KUKA KRL program: f1_Kuka_APT213T02S13.SRC

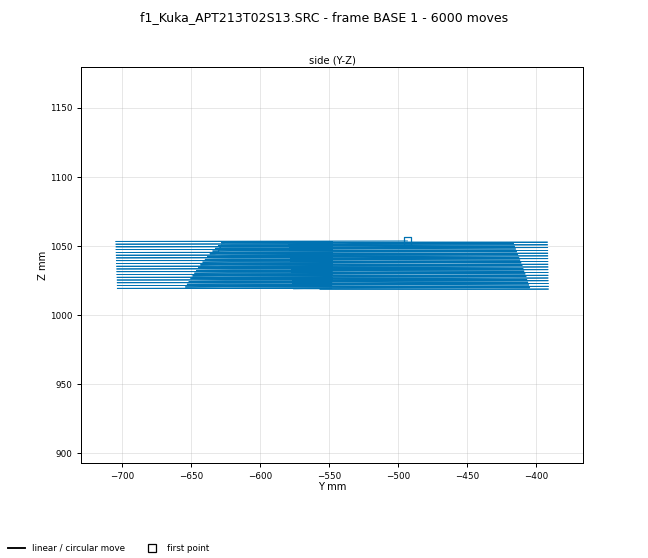
[picture p0: tool path of f1_Kuka_APT213T02S13.SRC in frame BASE 1, 6000 of 6001 moves have a stored position in this frame; points joined in program order, loops and branches not executed]
&ACCESS RVP
&REL 2
&PARAM TEMPLATE = C:\KRC\Roboter\Template\vorgabe
&PARAM EDITMASK = *
DEF f1_Kuka_APT213T02S13()


;FOLD INI;%{PE}%V3.2.0,%MKUKATPBASIS,%CINIT,%VCOMMON,%P
  ;FOLD BAS INI;%{E}%V3.2.0,%MKUKATPBASIS,%CINIT,%VINIT,%P
    GLOBAL INTERRUPT DECL 3 WHEN $STOPMESS==TRUE DO IR_STOPM ( )
    INTERRUPT ON 3
    BAS (#INITMOV,0 )
  ;ENDFOLD (BAS INI)
  ;FOLD USER INI;%{E}%V3.2.0,%MKUKATPUSER,%CINIT,%VINIT,%P
    ;Make your modifications here
  ;ENDFOLD (USER INI)
;ENDFOLD (INI)


;*** Make Null PTP Move
  PTP $pos_act

;*** Auto Load The Correct TOOL Data
  $tool=tool_data[2]

;*** Auto Load The Correct BASE Data
  $base=base_data[1]

  $ADVANCE = 5

;*** Restate Last Velocity
MMPM(30000.0)
SetRPM(8000)
LIN {X 0.196,Y -493.060,Z 1053.803,A 0.000,B 0.000,C 90.000,E1 180.573} C_DIS
LIN {X -0.057,Y -499.392,Z 1053.797,A 0.000,B 0.000,C 90.000,E1 179.542} C_DIS
LIN {X 0.076,Y -508.774,Z 1053.788,A 0.000,B 0.000,C 90.000,E1 177.879} C_DIS
LIN {X 0.040,Y -514.640,Z 1053.783,A 0.000,B 0.000,C 90.000,E1 176.846} C_DIS
LIN {X 0.239,Y -524.434,Z 1053.773,A 0.000,B 0.000,C 90.000,E1 175.065} C_DIS
LIN {X -0.105,Y -531.617,Z 1053.766,A 0.000,B 0.000,C 90.000,E1 173.799} C_DIS
LIN {X -0.076,Y -537.841,Z 1053.759,A 0.000,B 0.000,C 90.000,E1 172.648} C_DIS
LIN {X 0.196,Y -545.614,Z 1053.751,A 0.000,B 0.000,C 90.000,E1 171.197} C_DIS
LIN {X 0.075,Y -553.106,Z 1053.743,A 0.000,B 0.000,C 90.000,E1 169.803} C_DIS
LIN {X -0.212,Y -559.744,Z 1053.736,A 0.000,B 0.000,C 90.000,E1 168.578} C_DIS
LIN {X -0.238,Y -567.509,Z 1053.728,A 0.000,B 0.000,C 90.000,E1 167.061} C_DIS
LIN {X -0.052,Y -573.559,Z 1053.721,A 0.000,B 0.000,C 90.000,E1 165.811} C_DIS
LIN {X 0.098,Y -579.321,Z 1053.714,A 0.000,B 0.000,C 90.000,E1 164.574} C_DIS
LIN {X 0.012,Y -584.212,Z 1053.708,A 0.000,B 0.000,C 90.000,E1 163.504} C_DIS
LIN {X -0.002,Y -587.133,Z 1053.705,A 0.000,B 0.000,C 90.000,E1 162.834} C_DIS
LIN {X 0.006,Y -591.638,Z 1053.699,A 0.000,B 0.000,C 90.000,E1 161.764} C_DIS
LIN {X 0.001,Y -594.742,Z 1053.694,A 0.000,B 0.000,C 90.000,E1 160.967} C_DIS
LIN {X -0.165,Y -597.776,Z 1053.690,A 0.000,B 0.000,C 90.000,E1 160.188} C_DIS
LIN {X -0.189,Y -601.641,Z 1053.684,A 0.000,B 0.000,C 90.000,E1 159.135} C_DIS
LIN {X 0.188,Y -605.246,Z 1053.678,A 0.000,B 0.000,C 90.000,E1 158.050} C_DIS
LIN {X 0.000,Y -607.751,Z 1053.674,A 0.000,B 0.000,C 90.000,E1 157.283} C_DIS
LIN {X 0.082,Y -611.784,Z 1053.667,A 0.000,B 0.000,C 90.000,E1 155.973} C_DIS
LIN {X 0.223,Y -615.402,Z 1053.659,A 0.000,B 0.000,C 90.000,E1 154.665} C_DIS
LIN {X 0.159,Y -617.516,Z 1053.655,A 0.000,B 0.000,C 90.000,E1 153.896} C_DIS
LIN {X 0.107,Y -620.213,Z 1053.649,A 0.000,B 0.000,C 90.000,E1 152.871} C_DIS
LIN {X 0.086,Y -623.401,Z 1053.642,A 0.000,B 0.000,C 90.000,E1 151.591} C_DIS
LIN {X -0.142,Y -625.870,Z 1053.637,A 0.000,B 0.000,C 90.000,E1 150.589} C_DIS
LIN {X 0.226,Y -628.970,Z 1053.630,A 0.000,B 0.000,C 90.000,E1 149.282} C_DIS
LIN {X -0.091,Y -632.383,Z 1053.621,A 0.000,B 0.000,C 90.000,E1 147.788} C_DIS
LIN {X -0.338,Y -635.741,Z 1053.613,A 0.000,B 0.000,C 90.000,E1 146.294} C_DIS
LIN {X 0.223,Y -639.581,Z 1053.603,A 0.000,B 0.000,C 90.000,E1 144.482} C_DIS
LIN {X -0.163,Y -643.368,Z 1053.593,A 0.000,B 0.000,C 90.000,E1 142.763} C_DIS
LIN {X 0.016,Y -646.627,Z 1053.585,A 0.000,B 0.000,C 90.000,E1 141.251} C_DIS
LIN {X 0.163,Y -649.847,Z 1053.577,A 0.000,B 0.000,C 90.000,E1 139.747} C_DIS
LIN {X 0.329,Y -653.619,Z 1053.567,A 0.000,B 0.000,C 90.000,E1 138.000} C_DIS
LIN {X 0.123,Y -656.954,Z 1053.559,A 0.000,B 0.000,C 90.000,E1 136.539} C_DIS
LIN {X -0.151,Y -665.082,Z 1053.541,A 0.000,B 0.000,C 90.000,E1 133.380} C_DIS
LIN {X -0.134,Y -668.997,Z 1053.533,A 0.000,B 0.000,C 90.000,E1 131.919} C_DIS
LIN {X -0.029,Y -673.558,Z 1053.523,A 0.000,B 0.000,C 90.000,E1 130.216} C_DIS
LIN {X 0.230,Y -677.442,Z 1053.515,A 0.000,B 0.000,C 90.000,E1 128.749} C_DIS
LIN {X 0.011,Y -680.552,Z 1053.509,A 0.000,B 0.000,C 90.000,E1 127.569} C_DIS
LIN {X -0.011,Y -684.183,Z 1053.501,A 0.000,B 0.000,C 90.000,E1 126.137} C_DIS
LIN {X 0.008,Y -687.232,Z 1053.494,A 0.000,B 0.000,C 90.000,E1 124.945} C_DIS
LIN {X -0.079,Y -691.303,Z 1053.485,A 0.000,B 0.000,C 90.000,E1 123.293} C_DIS
LIN {X 0.024,Y -693.615,Z 1053.480,A 0.000,B 0.000,C 90.000,E1 122.339} C_DIS
LIN {X 0.155,Y -695.792,Z 1053.474,A 0.000,B 0.000,C 90.000,E1 121.386} C_DIS
LIN {X -0.048,Y -697.830,Z 1053.469,A 0.000,B 0.000,C 90.000,E1 120.463} C_DIS
LIN {X -0.222,Y -699.569,Z 1053.464,A 0.000,B 0.000,C 90.000,E1 119.539} C_DIS
LIN {X -0.034,Y -700.589,Z 1053.460,A 0.000,B 0.000,C 90.000,E1 118.821} C_DIS
LIN {X -0.015,Y -702.523,Z 1053.450,A 0.000,B 0.000,C 90.000,E1 116.950} C_DIS
LIN {X -0.150,Y -703.521,Z 1053.445,A 0.000,B 0.000,C 90.000,E1 116.027} C_DIS
LIN {X 0.042,Y -704.221,Z 1053.439,A 0.000,B 0.000,C 90.000,E1 115.079} C_DIS
LIN {X -0.324,Y -704.422,Z 1053.437,A 0.000,B 0.000,C 90.000,E1 114.643} C_DIS
LIN {X -0.045,Y -704.190,Z 1053.434,A 0.000,B 0.000,C 90.000,E1 114.155} C_DIS
LIN {X 0.240,Y -703.803,Z 1053.433,A 0.000,B 0.000,C 90.000,E1 113.898} C_DIS
LIN {X -0.123,Y -702.567,Z 1053.430,A 0.000,B 0.000,C 90.000,E1 113.462} C_DIS
LIN {X 0.017,Y -702.065,Z 1053.430,A 0.000,B 0.000,C 90.000,E1 113.334} C_DIS
LIN {X -0.357,Y -698.967,Z 1053.427,A 0.000,B 0.000,C 90.000,E1 112.898} C_DIS
LIN {X -0.223,Y -698.087,Z 1053.426,A 0.000,B 0.000,C 90.000,E1 112.770} C_DIS
LIN {X -0.093,Y -696.802,Z 1053.426,A 0.000,B 0.000,C 90.000,E1 112.642} C_DIS
LIN {X 0.037,Y -694.773,Z 1053.425,A 0.000,B 0.000,C 90.000,E1 112.514} C_DIS
LIN {X -0.179,Y -687.842,Z 1053.423,A 0.000,B 0.000,C 90.000,E1 112.206} C_DIS
LIN {X 0.203,Y -685.670,Z 1053.423,A 0.000,B 0.000,C 90.000,E1 112.099} C_DIS
LIN {X 0.017,Y -684.206,Z 1053.423,A 0.000,B 0.000,C 90.000,E1 112.078} C_DIS
LIN {X 0.020,Y -675.787,Z 1053.422,A 0.000,B 0.000,C 90.000,E1 111.972} C_DIS
LIN {X -0.030,Y -609.618,Z 1053.422,A 0.000,B 0.000,C 90.000,E1 111.972} C_DIS
LIN {X -0.052,Y -604.028,Z 1053.421,A 0.000,B 0.000,C 90.000,E1 111.770} C_DIS
LIN {X -0.108,Y -599.325,Z 1053.420,A 0.000,B 0.000,C 90.000,E1 111.535} C_DIS
LIN {X -0.008,Y -596.324,Z 1053.419,A 0.000,B 0.000,C 90.000,E1 111.354} C_DIS
LIN {X -0.148,Y -590.842,Z 1053.417,A 0.000,B 0.000,C 90.000,E1 110.972} C_DIS
LIN {X -0.111,Y -578.309,Z 1053.411,A 0.000,B 0.000,C 90.000,E1 109.939} C_DIS
LIN {X 0.049,Y -573.918,Z 1053.409,A 0.000,B 0.000,C 90.000,E1 109.577} C_DIS
LIN {X -0.218,Y -569.448,Z 1053.407,A 0.000,B 0.000,C 90.000,E1 109.268} C_DIS
LIN {X 0.182,Y -560.909,Z 1053.404,A 0.000,B 0.000,C 90.000,E1 108.725} C_DIS
LIN {X 0.205,Y -554.438,Z 1053.402,A 0.000,B 0.000,C 90.000,E1 108.362} C_DIS
LIN {X -0.142,Y -549.295,Z 1053.400,A 0.000,B 0.000,C 90.000,E1 108.055} C_DIS
LIN {X 0.269,Y -547.775,Z 1053.399,A 0.000,B 0.000,C 90.000,E1 107.819} C_DIS
LIN {X 0.228,Y -547.759,Z 1053.399,A 0.000,B 0.000,C 90.000,E1 107.819} C_DIS
LIN {X 0.214,Y -547.328,Z 1053.398,A 0.000,B 0.000,C 90.000,E1 107.583} C_DIS
LIN {X -0.058,Y -547.320,Z 1053.396,A 0.000,B 0.000,C 90.000,E1 107.330} C_DIS
LIN {X -0.165,Y -548.516,Z 1053.385,A 0.000,B 0.000,C 90.000,E1 105.371} C_DIS
LIN {X -0.133,Y -549.999,Z 1053.373,A 0.000,B 0.000,C 90.000,E1 103.119} C_DIS
LIN {X -0.195,Y -552.184,Z 1053.359,A 0.000,B 0.000,C 90.000,E1 100.602} C_DIS
LIN {X -0.117,Y -554.002,Z 1053.349,A 0.000,B 0.000,C 90.000,E1 98.916} C_DIS
LIN {X -0.209,Y -555.569,Z 1053.342,A 0.000,B 0.000,C 90.000,E1 97.530} C_DIS
LIN {X -0.268,Y -557.199,Z 1053.334,A 0.000,B 0.000,C 90.000,E1 96.144} C_DIS
LIN {X 0.123,Y -558.323,Z 1053.328,A 0.000,B 0.000,C 90.000,E1 94.992} C_DIS
LIN {X -0.032,Y -559.189,Z 1053.322,A 0.000,B 0.000,C 90.000,E1 93.898} C_DIS
LIN {X -0.218,Y -559.895,Z 1053.316,A 0.000,B 0.000,C 90.000,E1 92.808} C_DIS
LIN {X 0.165,Y -560.420,Z 1053.309,A 0.000,B 0.000,C 90.000,E1 91.661} C_DIS
LIN {X 0.171,Y -561.080,Z 1053.300,A 0.000,B 0.000,C 90.000,E1 90.000} C_DIS
LIN {X 0.094,Y -561.505,Z 1053.292,A 0.000,B 0.000,C 90.000,E1 88.625} C_DIS
LIN {X 0.259,Y -562.148,Z 1053.282,A 0.000,B 0.000,C 90.000,E1 86.674} C_DIS
LIN {X 0.211,Y -562.712,Z 1053.274,A 0.000,B 0.000,C 90.000,E1 85.298} C_DIS
LIN {X 0.266,Y -563.088,Z 1053.266,A 0.000,B 0.000,C 90.000,E1 83.913} C_DIS
LIN {X -0.139,Y -563.488,Z 1053.257,A 0.000,B 0.000,C 90.000,E1 82.299} C_DIS
LIN {X 0.087,Y -564.018,Z 1053.248,A 0.000,B 0.000,C 90.000,E1 80.622} C_DIS
LIN {X 0.184,Y -564.898,Z 1053.236,A 0.000,B 0.000,C 90.000,E1 78.409} C_DIS
LIN {X -0.089,Y -565.621,Z 1053.228,A 0.000,B 0.000,C 90.000,E1 77.061} C_DIS
LIN {X 0.052,Y -567.090,Z 1053.214,A 0.000,B 0.000,C 90.000,E1 74.574} C_DIS
LIN {X -0.267,Y -568.319,Z 1053.205,A 0.000,B 0.000,C 90.000,E1 72.960} C_DIS
LIN {X 0.117,Y -570.152,Z 1053.193,A 0.000,B 0.000,C 90.000,E1 70.732} C_DIS
LIN {X -0.132,Y -571.286,Z 1053.185,A 0.000,B 0.000,C 90.000,E1 69.390} C_DIS
LIN {X 0.206,Y -572.498,Z 1053.176,A 0.000,B 0.000,C 90.000,E1 67.720} C_DIS
LIN {X 0.043,Y -573.624,Z 1053.167,A 0.000,B 0.000,C 90.000,E1 66.102} C_DIS
LIN {X 0.086,Y -574.129,Z 1053.163,A 0.000,B 0.000,C 90.000,E1 65.281} C_DIS
LIN {X -0.175,Y -574.900,Z 1053.155,A 0.000,B 0.000,C 90.000,E1 63.948} C_DIS
LIN {X 0.081,Y -575.611,Z 1053.148,A 0.000,B 0.000,C 90.000,E1 62.564} C_DIS
LIN {X 0.211,Y -576.438,Z 1053.139,A 0.000,B 0.000,C 90.000,E1 60.923} C_DIS
LIN {X -0.134,Y -577.157,Z 1053.130,A 0.000,B 0.000,C 90.000,E1 59.331} C_DIS
LIN {X -0.155,Y -577.582,Z 1053.124,A 0.000,B 0.000,C 90.000,E1 58.250} C_DIS
LIN {X -0.169,Y -578.011,Z 1053.118,A 0.000,B 0.000,C 90.000,E1 57.168} C_DIS
LIN {X -0.025,Y -578.428,Z 1053.110,A 0.000,B 0.000,C 90.000,E1 55.801} C_DIS
LIN {X -0.195,Y -578.853,Z 1053.101,A 0.000,B 0.000,C 90.000,E1 54.196} C_DIS
LIN {X 0.133,Y -578.954,Z 1053.098,A 0.000,B 0.000,C 90.000,E1 53.623} C_DIS
LIN {X 0.143,Y -578.897,Z 1053.091,A 0.000,B 0.000,C 90.000,E1 52.271} C_DIS
LIN {X 0.339,Y -578.706,Z 1053.084,A 0.000,B 0.000,C 90.000,E1 51.170} C_DIS
LIN {X 0.245,Y -578.210,Z 1053.077,A 0.000,B 0.000,C 90.000,E1 49.828} C_DIS
LIN {X 0.139,Y -577.524,Z 1053.069,A 0.000,B 0.000,C 90.000,E1 48.485} C_DIS
LIN {X 0.253,Y -576.873,Z 1053.063,A 0.000,B 0.000,C 90.000,E1 47.391} C_DIS
LIN {X -0.058,Y -576.062,Z 1053.057,A 0.000,B 0.000,C 90.000,E1 46.338} C_DIS
LIN {X 0.322,Y -575.272,Z 1053.053,A 0.000,B 0.000,C 90.000,E1 45.486} C_DIS
LIN {X -0.007,Y -573.920,Z 1053.047,A 0.000,B 0.000,C 90.000,E1 44.433} C_DIS
LIN {X 0.058,Y -572.349,Z 1053.041,A 0.000,B 0.000,C 90.000,E1 43.338} C_DIS
LIN {X 0.104,Y -570.566,Z 1053.035,A 0.000,B 0.000,C 90.000,E1 42.243} C_DIS
LIN {X 0.306,Y -569.631,Z 1053.032,A 0.000,B 0.000,C 90.000,E1 41.676} C_DIS
LIN {X -0.072,Y -567.376,Z 1053.026,A 0.000,B 0.000,C 90.000,E1 40.620} C_DIS
LIN {X -0.270,Y -566.071,Z 1053.023,A 0.000,B 0.000,C 90.000,E1 40.092} C_DIS
LIN {X -0.011,Y -563.987,Z 1053.018,A 0.000,B 0.000,C 90.000,E1 39.241} C_DIS
LIN {X 0.201,Y -562.416,Z 1053.015,A 0.000,B 0.000,C 90.000,E1 38.669} C_DIS
LIN {X 0.059,Y -559.856,Z 1053.010,A 0.000,B 0.000,C 90.000,E1 37.855} C_DIS
LIN {X -0.094,Y -557.951,Z 1053.007,A 0.000,B 0.000,C 90.000,E1 37.317} C_DIS
LIN {X 0.165,Y -554.807,Z 1053.003,A 0.000,B 0.000,C 90.000,E1 36.457} C_DIS
LIN {X -0.063,Y -551.517,Z 1052.998,A 0.000,B 0.000,C 90.000,E1 35.644} C_DIS
LIN {X -0.205,Y -547.661,Z 1052.993,A 0.000,B 0.000,C 90.000,E1 34.818} C_DIS
LIN {X 0.371,Y -543.544,Z 1052.989,A 0.000,B 0.000,C 90.000,E1 33.913} C_DIS
LIN {X -0.136,Y -537.494,Z 1052.982,A 0.000,B 0.000,C 90.000,E1 32.832} C_DIS
LIN {X 0.030,Y -532.686,Z 1052.978,A 0.000,B 0.000,C 90.000,E1 31.957} C_DIS
LIN {X -0.005,Y -529.238,Z 1052.974,A 0.000,B 0.000,C 90.000,E1 31.386} C_DIS
LIN {X 0.107,Y -525.556,Z 1052.971,A 0.000,B 0.000,C 90.000,E1 30.797} C_DIS
LIN {X 0.033,Y -520.618,Z 1052.967,A 0.000,B 0.000,C 90.000,E1 30.079} C_DIS
LIN {X 0.175,Y -515.308,Z 1052.963,A 0.000,B 0.000,C 90.000,E1 29.333} C_DIS
LIN {X 0.185,Y -510.883,Z 1052.960,A 0.000,B 0.000,C 90.000,E1 28.743} C_DIS
LIN {X 0.163,Y -505.987,Z 1052.957,A 0.000,B 0.000,C 90.000,E1 28.153} C_DIS
LIN {X -0.021,Y -499.388,Z 1052.953,A 0.000,B 0.000,C 90.000,E1 27.436} C_DIS
LIN {X -0.034,Y -495.331,Z 1052.950,A 0.000,B 0.000,C 90.000,E1 27.001} C_DIS
LIN {X -0.074,Y -489.759,Z 1052.947,A 0.000,B 0.000,C 90.000,E1 26.437} C_DIS
LIN {X 0.284,Y -481.804,Z 1052.942,A 0.000,B 0.000,C 90.000,E1 25.591} C_DIS
LIN {X 0.123,Y -470.195,Z 1052.936,A 0.000,B 0.000,C 90.000,E1 24.515} C_DIS
LIN {X -0.206,Y -462.739,Z 1052.933,A 0.000,B 0.000,C 90.000,E1 23.898} C_DIS
LIN {X 0.077,Y -452.040,Z 1052.928,A 0.000,B 0.000,C 90.000,E1 22.950} C_DIS
LIN {X 0.152,Y -427.964,Z 1052.916,A 0.000,B 0.000,C 90.000,E1 20.791} C_DIS
LIN {X 0.092,Y -415.293,Z 1052.908,A 0.000,B 0.000,C 90.000,E1 19.504} C_DIS
LIN {X 0.041,Y -407.196,Z 1052.903,A 0.000,B 0.000,C 90.000,E1 18.598} C_DIS
LIN {X 0.054,Y -400.379,Z 1052.899,A 0.000,B 0.000,C 90.000,E1 17.764} C_DIS
LIN {X -0.100,Y -397.066,Z 1052.896,A 0.000,B 0.000,C 90.000,E1 17.330} C_DIS
LIN {X 0.132,Y -394.270,Z 1052.894,A 0.000,B 0.000,C 90.000,E1 16.804} C_DIS
LIN {X 0.017,Y -393.851,Z 1052.893,A 0.000,B 0.000,C 90.000,E1 16.732} C_DIS
LIN {X -0.007,Y -392.183,Z 1052.890,A 0.000,B 0.000,C 90.000,E1 16.205} C_DIS
LIN {X 0.069,Y -391.636,Z 1052.887,A 0.000,B 0.000,C 90.000,E1 15.662} C_DIS
LIN {X 0.051,Y -391.609,Z 1052.885,A 0.000,B 0.000,C 90.000,E1 15.300} C_DIS
LIN {X -0.008,Y -391.685,Z 1052.883,A 0.000,B 0.000,C 90.000,E1 14.954} C_DIS
LIN {X -0.032,Y -394.056,Z 1052.871,A 0.000,B 0.000,C 90.000,E1 12.827} C_DIS
LIN {X 0.152,Y -401.105,Z 1052.846,A 0.000,B 0.000,C 90.000,E1 8.219} C_DIS
LIN {X -0.012,Y -408.323,Z 1052.827,A 0.000,B 0.000,C 90.000,E1 4.759} C_DIS
LIN {X -0.045,Y -410.733,Z 1052.821,A 0.000,B 0.000,C 90.000,E1 3.726} C_DIS
LIN {X -0.056,Y -411.793,Z 1052.819,A 0.000,B 0.000,C 90.000,E1 3.383} C_DIS
LIN {X 0.189,Y -414.636,Z 1052.815,A 0.000,B 0.000,C 90.000,E1 2.751} C_DIS
LIN {X 0.192,Y -415.627,Z 1052.815,A 0.000,B 0.000,C 90.000,E1 2.579} C_DIS
LIN {X 0.196,Y -416.861,Z 1052.814,A 0.000,B 0.000,C 90.000,E1 2.407} C_DIS
LIN {X -0.001,Y -418.167,Z 1052.813,A 0.000,B 0.000,C 90.000,E1 2.293} C_DIS
LIN {X 0.066,Y -421.255,Z 1052.811,A 0.000,B 0.000,C 90.000,E1 2.007} C_DIS
LIN {X 0.157,Y -432.202,Z 1052.807,A 0.000,B 0.000,C 90.000,E1 1.260} C_DIS
LIN {X 0.086,Y -453.961,Z 1052.799,A 0.000,B 0.000,C 90.000,E1 359.885} C_DIS
LIN {X 0.178,Y -475.310,Z 1052.792,A 0.000,B 0.000,C 90.000,E1 358.568} C_DIS
LIN {X 0.220,Y -488.415,Z 1052.788,A 0.000,B 0.000,C 90.000,E1 357.764} C_DIS
LIN {X -0.109,Y -497.955,Z 1052.784,A 0.000,B 0.000,C 90.000,E1 357.192} C_DIS
LIN {X 0.259,Y -504.230,Z 1052.782,A 0.000,B 0.000,C 90.000,E1 356.731} C_DIS
LIN {X -0.042,Y -510.477,Z 1052.780,A 0.000,B 0.000,C 90.000,E1 356.331} C_DIS
LIN {X 0.082,Y -517.960,Z 1052.776,A 0.000,B 0.000,C 90.000,E1 355.755} C_DIS
LIN {X -0.053,Y -525.210,Z 1052.773,A 0.000,B 0.000,C 90.000,E1 355.179} C_DIS
LIN {X 0.092,Y -530.809,Z 1052.771,A 0.000,B 0.000,C 90.000,E1 354.666} C_DIS
LIN {X -0.239,Y -534.930,Z 1052.768,A 0.000,B 0.000,C 90.000,E1 354.318} C_DIS
LIN {X -0.030,Y -541.417,Z 1052.765,A 0.000,B 0.000,C 90.000,E1 353.628} C_DIS
LIN {X 0.136,Y -546.399,Z 1052.761,A 0.000,B 0.000,C 90.000,E1 353.053} C_DIS
LIN {X 0.061,Y -552.025,Z 1052.758,A 0.000,B 0.000,C 90.000,E1 352.356} C_DIS
LIN {X 0.213,Y -556.171,Z 1052.755,A 0.000,B 0.000,C 90.000,E1 351.781} C_DIS
LIN {X -0.078,Y -559.890,Z 1052.751,A 0.000,B 0.000,C 90.000,E1 351.254} C_DIS
LIN {X -0.119,Y -564.849,Z 1052.747,A 0.000,B 0.000,C 90.000,E1 350.443} C_DIS
LIN {X -0.028,Y -568.624,Z 1052.743,A 0.000,B 0.000,C 90.000,E1 349.746} C_DIS
LIN {X -0.273,Y -573.479,Z 1052.738,A 0.000,B 0.000,C 90.000,E1 348.814} C_DIS
LIN {X -0.228,Y -577.266,Z 1052.733,A 0.000,B 0.000,C 90.000,E1 347.993} C_DIS
LIN {X 0.312,Y -581.357,Z 1052.728,A 0.000,B 0.000,C 90.000,E1 346.992} C_DIS
LIN {X 0.106,Y -585.733,Z 1052.722,A 0.000,B 0.000,C 90.000,E1 345.936} C_DIS
LIN {X -0.214,Y -590.894,Z 1052.715,A 0.000,B 0.000,C 90.000,E1 344.629} C_DIS
LIN {X 0.118,Y -595.828,Z 1052.707,A 0.000,B 0.000,C 90.000,E1 343.268} C_DIS
LIN {X -0.146,Y -599.483,Z 1052.701,A 0.000,B 0.000,C 90.000,E1 342.236} C_DIS
LIN {X 0.218,Y -602.890,Z 1052.695,A 0.000,B 0.000,C 90.000,E1 341.148} C_DIS
LIN {X 0.060,Y -606.033,Z 1052.690,A 0.000,B 0.000,C 90.000,E1 340.115} C_DIS
LIN {X -0.117,Y -609.659,Z 1052.682,A 0.000,B 0.000,C 90.000,E1 338.827} C_DIS
LIN {X -0.197,Y -612.292,Z 1052.677,A 0.000,B 0.000,C 90.000,E1 337.794} C_DIS
LIN {X -0.017,Y -614.737,Z 1052.671,A 0.000,B 0.000,C 90.000,E1 336.741} C_DIS
LIN {X -0.120,Y -616.971,Z 1052.665,A 0.000,B 0.000,C 90.000,E1 335.717} C_DIS
LIN {X 0.133,Y -618.437,Z 1052.661,A 0.000,B 0.000,C 90.000,E1 334.921} C_DIS
LIN {X 0.082,Y -620.578,Z 1052.654,A 0.000,B 0.000,C 90.000,E1 333.640} C_DIS
LIN {X 0.068,Y -622.406,Z 1052.646,A 0.000,B 0.000,C 90.000,E1 332.359} C_DIS
LIN {X 0.370,Y -623.801,Z 1052.641,A 0.000,B 0.000,C 90.000,E1 331.307} C_DIS
LIN {X -0.155,Y -624.981,Z 1052.635,A 0.000,B 0.000,C 90.000,E1 330.333} C_DIS
LIN {X -0.352,Y -626.052,Z 1052.628,A 0.000,B 0.000,C 90.000,E1 329.076} C_DIS
LIN {X -0.015,Y -626.591,Z 1052.624,A 0.000,B 0.000,C 90.000,E1 328.280} C_DIS
LIN {X 0.133,Y -627.234,Z 1052.617,A 0.000,B 0.000,C 90.000,E1 326.993} C_DIS
LIN {X -0.229,Y -627.386,Z 1052.611,A 0.000,B 0.000,C 90.000,E1 326.008} C_DIS
LIN {X 0.283,Y -627.385,Z 1052.604,A 0.000,B 0.000,C 90.000,E1 324.689} C_DIS
LIN {X 0.279,Y -627.198,Z 1052.597,A 0.000,B 0.000,C 90.000,E1 323.417} C_DIS
LIN {X -0.026,Y -626.920,Z 1052.587,A 0.000,B 0.000,C 90.000,E1 321.662} C_DIS
LIN {X -0.336,Y -626.779,Z 1052.577,A 0.000,B 0.000,C 90.000,E1 319.908} C_DIS
LIN {X -0.055,Y -626.694,Z 1052.570,A 0.000,B 0.000,C 90.000,E1 318.609} C_DIS
LIN {X 0.225,Y -626.557,Z 1052.563,A 0.000,B 0.000,C 90.000,E1 317.310} C_DIS
LIN {X -0.089,Y -626.496,Z 1052.555,A 0.000,B 0.000,C 90.000,E1 315.810} C_DIS
LIN {X -0.097,Y -626.357,Z 1052.545,A 0.000,B 0.000,C 90.000,E1 314.028} C_DIS
LIN {X -0.287,Y -626.257,Z 1052.537,A 0.000,B 0.000,C 90.000,E1 312.771} C_DIS
LIN {X -0.349,Y -626.074,Z 1052.532,A 0.000,B 0.000,C 90.000,E1 311.757} C_DIS
LIN {X 0.115,Y -625.752,Z 1052.522,A 0.000,B 0.000,C 90.000,E1 309.930} C_DIS
LIN {X -0.228,Y -625.613,Z 1052.518,A 0.000,B 0.000,C 90.000,E1 309.197} C_DIS
LIN {X 0.302,Y -625.209,Z 1052.508,A 0.000,B 0.000,C 90.000,E1 307.363} C_DIS
LIN {X -0.233,Y -625.260,Z 1052.506,A 0.000,B 0.000,C 90.000,E1 307.156} C_DIS
LIN {X -0.051,Y -625.164,Z 1052.504,A 0.000,B 0.000,C 90.000,E1 306.629} C_DIS
LIN {X -0.082,Y -625.257,Z 1052.502,A 0.000,B 0.000,C 90.000,E1 306.377} C_DIS
LIN {X -0.271,Y -625.118,Z 1052.499,A 0.000,B 0.000,C 90.000,E1 305.884} C_DIS
LIN {X -0.120,Y -625.151,Z 1052.495,A 0.000,B 0.000,C 90.000,E1 305.105} C_DIS
LIN {X -0.310,Y -625.153,Z 1052.492,A 0.000,B 0.000,C 90.000,E1 304.612} C_DIS
LIN {X 0.028,Y -625.270,Z 1052.491,A 0.000,B 0.000,C 90.000,E1 304.326} C_DIS
LIN {X 0.015,Y -625.201,Z 1052.489,A 0.000,B 0.000,C 90.000,E1 304.072} C_DIS
LIN {X 0.160,Y -625.439,Z 1052.485,A 0.000,B 0.000,C 90.000,E1 303.293} C_DIS
LIN {X -0.039,Y -625.608,Z 1052.481,A 0.000,B 0.000,C 90.000,E1 302.546} C_DIS
LIN {X 0.097,Y -626.017,Z 1052.474,A 0.000,B 0.000,C 90.000,E1 301.258} C_DIS
LIN {X 0.109,Y -626.065,Z 1052.471,A 0.000,B 0.000,C 90.000,E1 300.747} C_DIS
LIN {X -0.096,Y -626.416,Z 1052.468,A 0.000,B 0.000,C 90.000,E1 300.256} C_DIS
LIN {X -0.086,Y -626.456,Z 1052.467,A 0.000,B 0.000,C 90.000,E1 300.001} C_DIS
LIN {X -0.062,Y -626.855,Z 1052.464,A 0.000,B 0.000,C 90.000,E1 299.489} C_DIS
LIN {X -0.259,Y -627.090,Z 1052.460,A 0.000,B 0.000,C 90.000,E1 298.743} C_DIS
LIN {X -0.227,Y -627.504,Z 1052.457,A 0.000,B 0.000,C 90.000,E1 298.231} C_DIS
LIN {X -0.127,Y -627.776,Z 1052.450,A 0.000,B 0.000,C 90.000,E1 296.950} C_DIS
LIN {X -0.083,Y -627.833,Z 1052.447,A 0.000,B 0.000,C 90.000,E1 296.437} C_DIS
LIN {X 0.002,Y -627.727,Z 1052.441,A 0.000,B 0.000,C 90.000,E1 295.412} C_DIS
LIN {X 0.079,Y -627.271,Z 1052.436,A 0.000,B 0.000,C 90.000,E1 294.387} C_DIS
LIN {X -0.116,Y -626.444,Z 1052.430,A 0.000,B 0.000,C 90.000,E1 293.387} C_DIS
LIN {X 0.255,Y -625.211,Z 1052.424,A 0.000,B 0.000,C 90.000,E1 292.333} C_DIS
LIN {X 0.029,Y -624.029,Z 1052.420,A 0.000,B 0.000,C 90.000,E1 291.589} C_DIS
LIN {X -0.205,Y -622.590,Z 1052.417,A 0.000,B 0.000,C 90.000,E1 291.099} C_DIS
LIN {X -0.213,Y -621.623,Z 1052.416,A 0.000,B 0.000,C 90.000,E1 290.844} C_DIS
LIN {X 0.117,Y -618.709,Z 1052.413,A 0.000,B 0.000,C 90.000,E1 290.301} C_DIS
LIN {X -0.152,Y -614.050,Z 1052.410,A 0.000,B 0.000,C 90.000,E1 289.812} C_DIS
LIN {X -0.041,Y -608.194,Z 1052.407,A 0.000,B 0.000,C 90.000,E1 289.322} C_DIS
LIN {X 0.075,Y -601.184,Z 1052.405,A 0.000,B 0.000,C 90.000,E1 288.906} C_DIS
LIN {X -0.108,Y -599.416,Z 1052.405,A 0.000,B 0.000,C 90.000,E1 288.833} C_DIS
LIN {X 0.029,Y -593.689,Z 1052.403,A 0.000,B 0.000,C 90.000,E1 288.598} C_DIS
LIN {X -0.035,Y -590.776,Z 1052.403,A 0.000,B 0.000,C 90.000,E1 288.471} C_DIS
LIN {X -0.036,Y -579.928,Z 1052.401,A 0.000,B 0.000,C 90.000,E1 288.127} C_DIS
LIN {X 0.084,Y -575.722,Z 1052.400,A 0.000,B 0.000,C 90.000,E1 288.000} C_DIS
LIN {X -0.126,Y -571.485,Z 1052.400,A 0.000,B 0.000,C 90.000,E1 287.928} C_DIS
LIN {X 0.154,Y -564.147,Z 1052.398,A 0.000,B 0.000,C 90.000,E1 287.692} C_DIS
LIN {X 0.036,Y -551.149,Z 1052.397,A 0.000,B 0.000,C 90.000,E1 287.402} C_DIS
LIN {X 0.186,Y -549.874,Z 1052.396,A 0.000,B 0.000,C 90.000,E1 287.347} C_DIS
LIN {X -0.023,Y -549.214,Z 1052.396,A 0.000,B 0.000,C 90.000,E1 287.330} C_DIS
LIN {X 0.193,Y -547.779,Z 1052.396,A 0.000,B 0.000,C 90.000,E1 287.166} C_DIS
LIN {X 0.129,Y -547.305,Z 1052.395,A 0.000,B 0.000,C 90.000,E1 286.985} C_DIS
LIN {X 0.080,Y -546.473,Z 1052.392,A 0.000,B 0.000,C 90.000,E1 286.567} C_DIS
LIN {X -0.219,Y -545.738,Z 1052.386,A 0.000,B 0.000,C 90.000,E1 285.552} C_DIS
LIN {X 0.069,Y -545.235,Z 1052.377,A 0.000,B 0.000,C 90.000,E1 283.828} C_DIS
LIN {X 0.113,Y -544.621,Z 1052.369,A 0.000,B 0.000,C 90.000,E1 282.411} C_DIS
LIN {X 0.024,Y -543.813,Z 1052.361,A 0.000,B 0.000,C 90.000,E1 281.007} C_DIS
LIN {X -0.098,Y -542.793,Z 1052.352,A 0.000,B 0.000,C 90.000,E1 279.321} C_DIS
LIN {X 0.216,Y -541.908,Z 1052.344,A 0.000,B 0.000,C 90.000,E1 277.871} C_DIS
LIN {X -0.094,Y -540.884,Z 1052.334,A 0.000,B 0.000,C 90.000,E1 276.201} C_DIS
LIN {X 0.108,Y -540.023,Z 1052.327,A 0.000,B 0.000,C 90.000,E1 274.759} C_DIS
LIN {X -0.264,Y -538.734,Z 1052.314,A 0.000,B 0.000,C 90.000,E1 272.522} C_DIS
LIN {X -0.171,Y -537.737,Z 1052.304,A 0.000,B 0.000,C 90.000,E1 270.802} C_DIS
LIN {X -0.103,Y -536.516,Z 1052.293,A 0.000,B 0.000,C 90.000,E1 268.797} C_DIS
LIN {X -0.066,Y -535.755,Z 1052.287,A 0.000,B 0.000,C 90.000,E1 267.650} C_DIS
LIN {X -0.007,Y -534.618,Z 1052.277,A 0.000,B 0.000,C 90.000,E1 265.927} C_DIS
LIN {X 0.059,Y -533.172,Z 1052.266,A 0.000,B 0.000,C 90.000,E1 263.913} C_DIS
LIN {X 0.052,Y -532.442,Z 1052.261,A 0.000,B 0.000,C 90.000,E1 263.053} C_DIS
LIN {X 0.172,Y -530.905,Z 1052.254,A 0.000,B 0.000,C 90.000,E1 261.602} C_DIS
LIN {X -0.216,Y -529.098,Z 1052.244,A 0.000,B 0.000,C 90.000,E1 259.916} C_DIS
LIN {X -0.184,Y -527.820,Z 1052.237,A 0.000,B 0.000,C 90.000,E1 258.757} C_DIS
LIN {X -0.056,Y -526.265,Z 1052.229,A 0.000,B 0.000,C 90.000,E1 257.297} C_DIS
LIN {X -0.189,Y -523.826,Z 1052.217,A 0.000,B 0.000,C 90.000,E1 254.991} C_DIS
LIN {X 0.258,Y -521.968,Z 1052.207,A 0.000,B 0.000,C 90.000,E1 253.196} C_DIS
LIN {X 0.023,Y -520.379,Z 1052.199,A 0.000,B 0.000,C 90.000,E1 251.764} C_DIS
LIN {X -0.089,Y -518.676,Z 1052.191,A 0.000,B 0.000,C 90.000,E1 250.315} C_DIS
LIN {X 0.076,Y -516.553,Z 1052.181,A 0.000,B 0.000,C 90.000,E1 248.539} C_DIS
LIN {X 0.128,Y -515.100,Z 1052.174,A 0.000,B 0.000,C 90.000,E1 247.358} C_DIS
LIN {X -0.070,Y -512.528,Z 1052.165,A 0.000,B 0.000,C 90.000,E1 245.613} C_DIS
LIN {X 0.133,Y -510.734,Z 1052.158,A 0.000,B 0.000,C 90.000,E1 244.409} C_DIS
LIN {X -0.055,Y -508.316,Z 1052.150,A 0.000,B 0.000,C 90.000,E1 242.948} C_DIS
LIN {X -0.139,Y -506.318,Z 1052.143,A 0.000,B 0.000,C 90.000,E1 241.769} C_DIS
LIN {X 0.125,Y -503.155,Z 1052.133,A 0.000,B 0.000,C 90.000,E1 239.950} C_DIS
LIN {X -0.011,Y -499.281,Z 1052.122,A 0.000,B 0.000,C 90.000,E1 237.867} C_DIS
LIN {X 0.295,Y -497.009,Z 1052.115,A 0.000,B 0.000,C 90.000,E1 236.628} C_DIS
LIN {X -0.122,Y -494.603,Z 1052.108,A 0.000,B 0.000,C 90.000,E1 235.468} C_DIS
LIN {X -0.006,Y -492.147,Z 1052.101,A 0.000,B 0.000,C 90.000,E1 234.242} C_DIS
LIN {X 0.021,Y -488.665,Z 1052.093,A 0.000,B 0.000,C 90.000,E1 232.718} C_DIS
LIN {X 0.132,Y -483.681,Z 1052.081,A 0.000,B 0.000,C 90.000,E1 230.561} C_DIS
LIN {X 0.001,Y -479.612,Z 1052.071,A 0.000,B 0.000,C 90.000,E1 228.728} C_DIS
LIN {X 0.254,Y -476.413,Z 1052.062,A 0.000,B 0.000,C 90.000,E1 227.148} C_DIS
LIN {X -0.022,Y -471.997,Z 1052.050,A 0.000,B 0.000,C 90.000,E1 225.000} C_DIS
LIN {X 0.095,Y -468.875,Z 1052.041,A 0.000,B 0.000,C 90.000,E1 223.419} C_DIS
LIN {X -0.095,Y -465.068,Z 1052.031,A 0.000,B 0.000,C 90.000,E1 221.553} C_DIS
LIN {X -0.227,Y -463.145,Z 1052.026,A 0.000,B 0.000,C 90.000,E1 220.620} C_DIS
LIN {X 0.137,Y -459.104,Z 1052.015,A 0.000,B 0.000,C 90.000,E1 218.669} C_DIS
LIN {X -0.079,Y -454.488,Z 1052.003,A 0.000,B 0.000,C 90.000,E1 216.457} C_DIS
LIN {X 0.159,Y -451.146,Z 1051.994,A 0.000,B 0.000,C 90.000,E1 214.818} C_DIS
LIN {X -0.258,Y -448.446,Z 1051.986,A 0.000,B 0.000,C 90.000,E1 213.579} C_DIS
LIN {X -0.098,Y -445.807,Z 1051.979,A 0.000,B 0.000,C 90.000,E1 212.260} C_DIS
LIN {X 0.153,Y -442.982,Z 1051.972,A 0.000,B 0.000,C 90.000,E1 210.924} C_DIS
LIN {X 0.184,Y -439.389,Z 1051.963,A 0.000,B 0.000,C 90.000,E1 209.283} C_DIS
LIN {X -0.012,Y -434.457,Z 1051.950,A 0.000,B 0.000,C 90.000,E1 207.001} C_DIS
LIN {X 0.034,Y -431.706,Z 1051.943,A 0.000,B 0.000,C 90.000,E1 205.668} C_DIS
LIN {X 0.182,Y -425.713,Z 1051.926,A 0.000,B 0.000,C 90.000,E1 202.642} C_DIS
LIN {X 0.192,Y -420.191,Z 1051.907,A 0.000,B 0.000,C 90.000,E1 199.268} C_DIS
LIN {X 0.109,Y -418.046,Z 1051.898,A 0.000,B 0.000,C 90.000,E1 197.583} C_DIS
LIN {X -0.017,Y -416.692,Z 1051.888,A 0.000,B 0.000,C 90.000,E1 195.898} C_DIS
LIN {X -0.182,Y -416.301,Z 1051.883,A 0.000,B 0.000,C 90.000,E1 194.898} C_DIS
LIN {X 0.012,Y -416.526,Z 1051.879,A 0.000,B 0.000,C 90.000,E1 194.189} C_DIS
LIN {X -0.198,Y -417.088,Z 1051.875,A 0.000,B 0.000,C 90.000,E1 193.536} C_DIS
LIN {X -0.002,Y -418.186,Z 1051.871,A 0.000,B 0.000,C 90.000,E1 192.827} C_DIS
LIN {X 0.209,Y -420.009,Z 1051.868,A 0.000,B 0.000,C 90.000,E1 192.119} C_DIS
LIN {X -0.141,Y -421.095,Z 1051.866,A 0.000,B 0.000,C 90.000,E1 191.827} C_DIS
LIN {X 0.000,Y -424.140,Z 1051.862,A 0.000,B 0.000,C 90.000,E1 191.130} C_DIS
LIN {X -0.231,Y -427.704,Z 1051.858,A 0.000,B 0.000,C 90.000,E1 190.489} C_DIS
LIN {X 0.087,Y -433.767,Z 1051.853,A 0.000,B 0.000,C 90.000,E1 189.443} C_DIS
LIN {X -0.079,Y -444.587,Z 1051.843,A 0.000,B 0.000,C 90.000,E1 187.814} C_DIS
LIN {X 0.139,Y -453.538,Z 1051.836,A 0.000,B 0.000,C 90.000,E1 186.486} C_DIS
LIN {X 0.096,Y -463.432,Z 1051.828,A 0.000,B 0.000,C 90.000,E1 185.049} C_DIS
LIN {X -0.158,Y -469.687,Z 1051.823,A 0.000,B 0.000,C 90.000,E1 184.131} C_DIS
LIN {X 0.132,Y -475.708,Z 1051.818,A 0.000,B 0.000,C 90.000,E1 183.154} C_DIS
LIN {X -0.013,Y -484.438,Z 1051.810,A 0.000,B 0.000,C 90.000,E1 181.776} C_DIS
LIN {X -0.215,Y -491.852,Z 1051.803,A 0.000,B 0.000,C 90.000,E1 180.573} C_DIS
LIN {X 0.192,Y -499.138,Z 1051.796,A 0.000,B 0.000,C 90.000,E1 179.312} C_DIS
LIN {X 0.121,Y -507.768,Z 1051.788,A 0.000,B 0.000,C 90.000,E1 177.822} C_DIS
LIN {X 0.074,Y -513.711,Z 1051.782,A 0.000,B 0.000,C 90.000,E1 176.788} C_DIS
LIN {X 0.199,Y -525.173,Z 1051.771,A 0.000,B 0.000,C 90.000,E1 174.723} C_DIS
LIN {X -0.083,Y -532.375,Z 1051.764,A 0.000,B 0.000,C 90.000,E1 173.451} C_DIS
LIN {X 0.234,Y -537.830,Z 1051.758,A 0.000,B 0.000,C 90.000,E1 172.413} C_DIS
LIN {X 0.162,Y -544.879,Z 1051.751,A 0.000,B 0.000,C 90.000,E1 171.141} C_DIS
LIN {X -0.237,Y -553.135,Z 1051.742,A 0.000,B 0.000,C 90.000,E1 169.634} C_DIS
LIN {X -0.275,Y -559.065,Z 1051.736,A 0.000,B 0.000,C 90.000,E1 168.522} C_DIS
LIN {X -0.191,Y -566.914,Z 1051.728,A 0.000,B 0.000,C 90.000,E1 166.992} C_DIS
LIN {X -0.031,Y -572.333,Z 1051.722,A 0.000,B 0.000,C 90.000,E1 165.880} C_DIS
LIN {X 0.243,Y -578.170,Z 1051.715,A 0.000,B 0.000,C 90.000,E1 164.629} C_DIS
LIN {X 0.233,Y -582.539,Z 1051.710,A 0.000,B 0.000,C 90.000,E1 163.685} C_DIS
LIN {X 0.287,Y -584.966,Z 1051.707,A 0.000,B 0.000,C 90.000,E1 163.142} C_DIS
LIN {X -0.295,Y -589.576,Z 1051.701,A 0.000,B 0.000,C 90.000,E1 162.127} C_DIS
LIN {X 0.237,Y -592.789,Z 1051.696,A 0.000,B 0.000,C 90.000,E1 161.275} C_DIS
LIN {X -0.059,Y -596.891,Z 1051.690,A 0.000,B 0.000,C 90.000,E1 160.242} C_DIS
LIN {X -0.303,Y -600.809,Z 1051.684,A 0.000,B 0.000,C 90.000,E1 159.209} C_DIS
LIN {X 0.280,Y -604.453,Z 1051.679,A 0.000,B 0.000,C 90.000,E1 158.103} C_DIS
LIN {X -0.147,Y -607.012,Z 1051.674,A 0.000,B 0.000,C 90.000,E1 157.358} C_DIS
LIN {X -0.085,Y -611.062,Z 1051.667,A 0.000,B 0.000,C 90.000,E1 156.049} C_DIS
LIN {X 0.299,Y -614.776,Z 1051.660,A 0.000,B 0.000,C 90.000,E1 154.717} C_DIS
LIN {X -0.059,Y -617.565,Z 1051.654,A 0.000,B 0.000,C 90.000,E1 153.717} C_DIS
LIN {X -0.105,Y -619.589,Z 1051.650,A 0.000,B 0.000,C 90.000,E1 152.948} C_DIS
LIN {X 0.153,Y -622.800,Z 1051.643,A 0.000,B 0.000,C 90.000,E1 151.641} C_DIS
LIN {X 0.156,Y -624.704,Z 1051.638,A 0.000,B 0.000,C 90.000,E1 150.873} C_DIS
LIN {X -0.044,Y -627.842,Z 1051.631,A 0.000,B 0.000,C 90.000,E1 149.616} C_DIS
LIN {X 0.151,Y -631.279,Z 1051.623,A 0.000,B 0.000,C 90.000,E1 148.074} C_DIS
LIN {X -0.142,Y -634.099,Z 1051.616,A 0.000,B 0.000,C 90.000,E1 146.834} C_DIS
LIN {X 0.120,Y -636.336,Z 1051.610,A 0.000,B 0.000,C 90.000,E1 145.801} C_DIS
LIN {X -0.216,Y -639.640,Z 1051.602,A 0.000,B 0.000,C 90.000,E1 144.322} C_DIS
LIN {X 0.019,Y -642.912,Z 1051.593,A 0.000,B 0.000,C 90.000,E1 142.798} C_DIS
LIN {X 0.093,Y -646.741,Z 1051.584,A 0.000,B 0.000,C 90.000,E1 141.045} C_DIS
LIN {X -0.192,Y -649.462,Z 1051.577,A 0.000,B 0.000,C 90.000,E1 139.828} C_DIS
LIN {X -0.039,Y -653.256,Z 1051.567,A 0.000,B 0.000,C 90.000,E1 138.081} C_DIS
LIN {X -0.289,Y -657.181,Z 1051.558,A 0.000,B 0.000,C 90.000,E1 136.377} C_DIS
LIN {X -0.065,Y -664.773,Z 1051.541,A 0.000,B 0.000,C 90.000,E1 133.419} C_DIS
LIN {X -0.091,Y -668.704,Z 1051.533,A 0.000,B 0.000,C 90.000,E1 131.962} C_DIS
LIN {X 0.073,Y -673.301,Z 1051.524,A 0.000,B 0.000,C 90.000,E1 130.253} C_DIS
LIN {X -0.186,Y -677.193,Z 1051.516,A 0.000,B 0.000,C 90.000,E1 128.830} C_DIS
LIN {X 0.149,Y -680.923,Z 1051.508,A 0.000,B 0.000,C 90.000,E1 127.363} C_DIS
LIN {X 0.118,Y -683.951,Z 1051.501,A 0.000,B 0.000,C 90.000,E1 126.171} C_DIS
LIN {X 0.166,Y -687.589,Z 1051.493,A 0.000,B 0.000,C 90.000,E1 124.739} C_DIS
LIN {X 0.089,Y -691.708,Z 1051.484,A 0.000,B 0.000,C 90.000,E1 123.086} C_DIS
LIN {X -0.158,Y -694.531,Z 1051.477,A 0.000,B 0.000,C 90.000,E1 121.926} C_DIS
LIN {X 0.227,Y -697.187,Z 1051.471,A 0.000,B 0.000,C 90.000,E1 120.718} C_DIS
LIN {X 0.042,Y -698.966,Z 1051.466,A 0.000,B 0.000,C 90.000,E1 119.795} C_DIS
LIN {X -0.122,Y -700.400,Z 1051.460,A 0.000,B 0.000,C 90.000,E1 118.871} C_DIS
LIN {X 0.345,Y -701.401,Z 1051.455,A 0.000,B 0.000,C 90.000,E1 117.897} C_DIS
LIN {X 0.092,Y -703.194,Z 1051.446,A 0.000,B 0.000,C 90.000,E1 116.283} C_DIS
LIN {X -0.003,Y -703.798,Z 1051.442,A 0.000,B 0.000,C 90.000,E1 115.591} C_DIS
LIN {X 0.196,Y -704.385,Z 1051.437,A 0.000,B 0.000,C 90.000,E1 114.643} C_DIS
LIN {X -0.167,Y -704.152,Z 1051.434,A 0.000,B 0.000,C 90.000,E1 114.207} C_DIS
LIN {X 0.117,Y -703.849,Z 1051.433,A 0.000,B 0.000,C 90.000,E1 113.951} C_DIS
LIN {X -0.248,Y -702.657,Z 1051.431,A 0.000,B 0.000,C 90.000,E1 113.515} C_DIS
LIN {X 0.030,Y -701.564,Z 1051.429,A 0.000,B 0.000,C 90.000,E1 113.259} C_DIS
LIN {X 0.295,Y -698.477,Z 1051.427,A 0.000,B 0.000,C 90.000,E1 112.770} C_DIS
LIN {X -0.218,Y -697.371,Z 1051.426,A 0.000,B 0.000,C 90.000,E1 112.695} C_DIS
LIN {X -0.355,Y -695.682,Z 1051.425,A 0.000,B 0.000,C 90.000,E1 112.589} C_DIS
LIN {X 0.070,Y -688.442,Z 1051.423,A 0.000,B 0.000,C 90.000,E1 112.206} C_DIS
LIN {X -0.204,Y -686.384,Z 1051.423,A 0.000,B 0.000,C 90.000,E1 112.153} C_DIS
LIN {X -0.218,Y -683.142,Z 1051.423,A 0.000,B 0.000,C 90.000,E1 112.078} C_DIS
LIN {X -0.009,Y -676.098,Z 1051.422,A 0.000,B 0.000,C 90.000,E1 111.972} C_DIS
LIN {X -0.066,Y -609.859,Z 1051.422,A 0.000,B 0.000,C 90.000,E1 111.972} C_DIS
LIN {X -0.229,Y -603.902,Z 1051.421,A 0.000,B 0.000,C 90.000,E1 111.770} C_DIS
LIN {X 0.124,Y -597.551,Z 1051.419,A 0.000,B 0.000,C 90.000,E1 111.408} C_DIS
LIN {X -0.029,Y -592.038,Z 1051.417,A 0.000,B 0.000,C 90.000,E1 111.046} C_DIS
LIN {X 0.344,Y -577.393,Z 1051.410,A 0.000,B 0.000,C 90.000,E1 109.812} C_DIS
LIN {X -0.071,Y -572.864,Z 1051.408,A 0.000,B 0.000,C 90.000,E1 109.504} C_DIS
LIN {X 0.091,Y -569.953,Z 1051.407,A 0.000,B 0.000,C 90.000,E1 109.268} C_DIS
LIN {X 0.166,Y -563.233,Z 1051.405,A 0.000,B 0.000,C 90.000,E1 108.852} C_DIS
LIN {X 0.184,Y -553.612,Z 1051.402,A 0.000,B 0.000,C 90.000,E1 108.308} C_DIS
LIN {X 0.207,Y -549.783,Z 1051.401,A 0.000,B 0.000,C 90.000,E1 108.055} C_DIS
LIN {X -0.244,Y -548.800,Z 1051.400,A 0.000,B 0.000,C 90.000,E1 108.000} C_DIS
LIN {X 0.272,Y -547.787,Z 1051.399,A 0.000,B 0.000,C 90.000,E1 107.819} C_DIS
LIN {X 0.230,Y -547.765,Z 1051.399,A 0.000,B 0.000,C 90.000,E1 107.819} C_DIS
LIN {X -0.287,Y -547.286,Z 1051.398,A 0.000,B 0.000,C 90.000,E1 107.583} C_DIS
LIN {X -0.283,Y -548.639,Z 1051.384,A 0.000,B 0.000,C 90.000,E1 105.190} C_DIS
LIN {X -0.035,Y -550.595,Z 1051.369,A 0.000,B 0.000,C 90.000,E1 102.355} C_DIS
LIN {X 0.060,Y -553.578,Z 1051.352,A 0.000,B 0.000,C 90.000,E1 99.265} C_DIS
LIN {X 0.209,Y -555.758,Z 1051.341,A 0.000,B 0.000,C 90.000,E1 97.296} C_DIS
LIN {X 0.024,Y -557.075,Z 1051.334,A 0.000,B 0.000,C 90.000,E1 96.201} C_DIS
LIN {X -0.143,Y -558.221,Z 1051.328,A 0.000,B 0.000,C 90.000,E1 95.106} C_DIS
LIN {X 0.256,Y -559.129,Z 1051.322,A 0.000,B 0.000,C 90.000,E1 93.955} C_DIS
LIN {X 0.158,Y -559.975,Z 1051.314,A 0.000,B 0.000,C 90.000,E1 92.579} C_DIS
LIN {X -0.110,Y -560.362,Z 1051.310,A 0.000,B 0.000,C 90.000,E1 91.776} C_DIS
LIN {X -0.106,Y -561.023,Z 1051.301,A 0.000,B 0.000,C 90.000,E1 90.115} C_DIS
LIN {X -0.183,Y -561.454,Z 1051.293,A 0.000,B 0.000,C 90.000,E1 88.740} C_DIS
LIN {X -0.146,Y -561.976,Z 1051.284,A 0.000,B 0.000,C 90.000,E1 87.078} C_DIS
LIN {X -0.067,Y -562.621,Z 1051.275,A 0.000,B 0.000,C 90.000,E1 85.412} C_DIS
LIN {X -0.072,Y -563.003,Z 1051.267,A 0.000,B 0.000,C 90.000,E1 84.033} C_DIS
LIN {X -0.094,Y -563.276,Z 1051.261,A 0.000,B 0.000,C 90.000,E1 82.932} C_DIS
LIN {X 0.211,Y -563.845,Z 1051.250,A 0.000,B 0.000,C 90.000,E1 80.971} C_DIS
LIN {X -0.083,Y -564.796,Z 1051.236,A 0.000,B 0.000,C 90.000,E1 78.522} C_DIS
LIN {X 0.199,Y -565.512,Z 1051.229,A 0.000,B 0.000,C 90.000,E1 77.117} C_DIS
LIN {X -0.205,Y -566.970,Z 1051.215,A 0.000,B 0.000,C 90.000,E1 74.685} C_DIS
LIN {X 0.025,Y -568.214,Z 1051.206,A 0.000,B 0.000,C 90.000,E1 73.015} C_DIS
LIN {X -0.312,Y -570.032,Z 1051.193,A 0.000,B 0.000,C 90.000,E1 70.859} C_DIS
LIN {X 0.169,Y -571.167,Z 1051.186,A 0.000,B 0.000,C 90.000,E1 69.444} C_DIS
LIN {X -0.237,Y -572.354,Z 1051.177,A 0.000,B 0.000,C 90.000,E1 67.847} C_DIS
LIN {X 0.120,Y -573.477,Z 1051.168,A 0.000,B 0.000,C 90.000,E1 66.177} C_DIS
LIN {X 0.157,Y -573.991,Z 1051.163,A 0.000,B 0.000,C 90.000,E1 65.357} C_DIS
LIN {X -0.113,Y -574.741,Z 1051.156,A 0.000,B 0.000,C 90.000,E1 64.024} C_DIS
LIN {X -0.113,Y -575.448,Z 1051.148,A 0.000,B 0.000,C 90.000,E1 62.666} C_DIS
LIN {X -0.250,Y -576.235,Z 1051.139,A 0.000,B 0.000,C 90.000,E1 61.051} C_DIS
LIN {X -0.101,Y -576.999,Z 1051.130,A 0.000,B 0.000,C 90.000,E1 59.410} C_DIS
LIN {X 0.028,Y -577.339,Z 1051.125,A 0.000,B 0.000,C 90.000,E1 58.584} C_DIS
LIN {X -0.147,Y -577.846,Z 1051.118,A 0.000,B 0.000,C 90.000,E1 57.248} C_DIS
LIN {X 0.148,Y -578.307,Z 1051.109,A 0.000,B 0.000,C 90.000,E1 55.595} C_DIS
LIN {X -0.188,Y -578.646,Z 1051.101,A 0.000,B 0.000,C 90.000,E1 54.276} C_DIS
LIN {X 0.299,Y -578.758,Z 1051.097,A 0.000,B 0.000,C 90.000,E1 53.417} C_DIS
LIN {X -0.155,Y -578.675,Z 1051.089,A 0.000,B 0.000,C 90.000,E1 52.110} C_DIS
LIN {X -0.120,Y -578.515,Z 1051.085,A 0.000,B 0.000,C 90.000,E1 51.295} C_DIS
LIN {X 0.076,Y -578.128,Z 1051.079,A 0.000,B 0.000,C 90.000,E1 50.194} C_DIS
LIN {X -0.028,Y -577.485,Z 1051.071,A 0.000,B 0.000,C 90.000,E1 48.852} C_DIS
LIN {X 0.089,Y -576.842,Z 1051.065,A 0.000,B 0.000,C 90.000,E1 47.757} C_DIS
LIN {X -0.195,Y -576.080,Z 1051.059,A 0.000,B 0.000,C 90.000,E1 46.701} C_DIS
LIN {X 0.297,Y -575.061,Z 1051.053,A 0.000,B 0.000,C 90.000,E1 45.567} C_DIS
LIN {X 0.252,Y -574.108,Z 1051.049,A 0.000,B 0.000,C 90.000,E1 44.757} C_DIS
LIN {X -0.096,Y -572.540,Z 1051.043,A 0.000,B 0.000,C 90.000,E1 43.704} C_DIS
LIN {X -0.052,Y -570.791,Z 1051.037,A 0.000,B 0.000,C 90.000,E1 42.609} C_DIS
LIN {X 0.271,Y -569.372,Z 1051.032,A 0.000,B 0.000,C 90.000,E1 41.757} C_DIS
LIN {X -0.109,Y -567.103,Z 1051.026,A 0.000,B 0.000,C 90.000,E1 40.701} C_DIS
LIN {X -0.309,Y -565.814,Z 1051.023,A 0.000,B 0.000,C 90.000,E1 40.172} C_DIS
LIN {X -0.050,Y -563.697,Z 1051.018,A 0.000,B 0.000,C 90.000,E1 39.322} C_DIS
LIN {X 0.160,Y -562.126,Z 1051.015,A 0.000,B 0.000,C 90.000,E1 38.749} C_DIS
LIN {X 0.110,Y -558.645,Z 1051.009,A 0.000,B 0.000,C 90.000,E1 37.649} C_DIS
LIN {X 0.036,Y -555.581,Z 1051.005,A 0.000,B 0.000,C 90.000,E1 36.824} C_DIS
LIN {X -0.110,Y -551.120,Z 1050.998,A 0.000,B 0.000,C 90.000,E1 35.724} C_DIS
LIN {X -0.252,Y -547.315,Z 1050.994,A 0.000,B 0.000,C 90.000,E1 34.898} C_DIS
LIN {X -0.127,Y -543.166,Z 1050.989,A 0.000,B 0.000,C 90.000,E1 34.040} C_DIS
LIN {X -0.046,Y -537.893,Z 1050.984,A 0.000,B 0.000,C 90.000,E1 33.038} C_DIS
LIN {X -0.327,Y -533.112,Z 1050.979,A 0.000,B 0.000,C 90.000,E1 32.212} C_DIS
LIN {X -0.057,Y -528.801,Z 1050.975,A 0.000,B 0.000,C 90.000,E1 31.465} C_DIS
LIN {X 0.054,Y -525.147,Z 1050.972,A 0.000,B 0.000,C 90.000,E1 30.875} C_DIS
LIN {X -0.310,Y -521.224,Z 1050.968,A 0.000,B 0.000,C 90.000,E1 30.335} C_DIS
LIN {X -0.249,Y -517.070,Z 1050.965,A 0.000,B 0.000,C 90.000,E1 29.745} C_DIS
LIN {X -0.144,Y -511.586,Z 1050.961,A 0.000,B 0.000,C 90.000,E1 28.999} C_DIS
LIN {X 0.108,Y -505.536,Z 1050.957,A 0.000,B 0.000,C 90.000,E1 28.231} C_DIS
LIN {X 0.088,Y -500.283,Z 1050.954,A 0.000,B 0.000,C 90.000,E1 27.641} C_DIS
LIN {X -0.080,Y -494.880,Z 1050.950,A 0.000,B 0.000,C 90.000,E1 27.078} C_DIS
LIN {X -0.100,Y -486.564,Z 1050.946,A 0.000,B 0.000,C 90.000,E1 26.232} C_DIS
LIN {X -0.031,Y -480.968,Z 1050.943,A 0.000,B 0.000,C 90.000,E1 25.668} C_DIS
LIN {X 0.009,Y -470.991,Z 1050.937,A 0.000,B 0.000,C 90.000,E1 24.719} C_DIS
LIN {X 0.135,Y -461.942,Z 1050.933,A 0.000,B 0.000,C 90.000,E1 23.898} C_DIS
LIN {X -0.164,Y -451.218,Z 1050.928,A 0.000,B 0.000,C 90.000,E1 23.025} C_DIS
LIN {X 0.105,Y -427.467,Z 1050.916,A 0.000,B 0.000,C 90.000,E1 20.865} C_DIS
LIN {X -0.083,Y -417.517,Z 1050.910,A 0.000,B 0.000,C 90.000,E1 19.885} C_DIS
LIN {X 0.249,Y -407.909,Z 1050.905,A 0.000,B 0.000,C 90.000,E1 18.779} C_DIS
LIN {X -0.007,Y -399.766,Z 1050.899,A 0.000,B 0.000,C 90.000,E1 17.819} C_DIS
LIN {X -0.015,Y -396.303,Z 1050.896,A 0.000,B 0.000,C 90.000,E1 17.330} C_DIS
LIN {X 0.202,Y -393.928,Z 1050.894,A 0.000,B 0.000,C 90.000,E1 16.858} C_DIS
LIN {X -0.014,Y -393.344,Z 1050.893,A 0.000,B 0.000,C 90.000,E1 16.732} C_DIS
LIN {X -0.216,Y -391.896,Z 1050.890,A 0.000,B 0.000,C 90.000,E1 16.205} C_DIS
LIN {X 0.184,Y -391.522,Z 1050.886,A 0.000,B 0.000,C 90.000,E1 15.481} C_DIS
LIN {X 0.201,Y -391.854,Z 1050.882,A 0.000,B 0.000,C 90.000,E1 14.773} C_DIS
LIN {X 0.001,Y -398.414,Z 1050.855,A 0.000,B 0.000,C 90.000,E1 9.849} C_DIS
LIN {X 0.193,Y -406.422,Z 1050.831,A 0.000,B 0.000,C 90.000,E1 5.625} C_DIS
LIN {X 0.145,Y -411.610,Z 1050.819,A 0.000,B 0.000,C 90.000,E1 3.383} C_DIS
LIN {X -0.043,Y -414.018,Z 1050.816,A 0.000,B 0.000,C 90.000,E1 2.865} C_DIS
LIN {X -0.044,Y -414.820,Z 1050.815,A 0.000,B 0.000,C 90.000,E1 2.694} C_DIS
LIN {X 0.002,Y -417.530,Z 1050.813,A 0.000,B 0.000,C 90.000,E1 2.293} C_DIS
LIN {X -0.178,Y -420.919,Z 1050.811,A 0.000,B 0.000,C 90.000,E1 2.007} C_DIS
LIN {X 0.057,Y -422.653,Z 1050.810,A 0.000,B 0.000,C 90.000,E1 1.835} C_DIS
LIN {X -0.160,Y -438.154,Z 1050.805,A 0.000,B 0.000,C 90.000,E1 0.859} C_DIS
LIN {X -0.199,Y -456.403,Z 1050.798,A 0.000,B 0.000,C 90.000,E1 359.714} C_DIS
LIN {X 0.222,Y -474.372,Z 1050.792,A 0.000,B 0.000,C 90.000,E1 358.568} C_DIS
LIN {X 0.155,Y -485.851,Z 1050.788,A 0.000,B 0.000,C 90.000,E1 357.879} C_DIS
LIN {X -0.227,Y -493.883,Z 1050.786,A 0.000,B 0.000,C 90.000,E1 357.421} C_DIS
LIN {X -0.089,Y -503.310,Z 1050.782,A 0.000,B 0.000,C 90.000,E1 356.788} C_DIS
LIN {X -0.256,Y -510.951,Z 1050.779,A 0.000,B 0.000,C 90.000,E1 356.274} C_DIS
LIN {X -0.040,Y -518.334,Z 1050.776,A 0.000,B 0.000,C 90.000,E1 355.698} C_DIS
LIN {X -0.052,Y -525.420,Z 1050.773,A 0.000,B 0.000,C 90.000,E1 355.122} C_DIS
LIN {X 0.029,Y -532.421,Z 1050.769,A 0.000,B 0.000,C 90.000,E1 354.489} C_DIS
LIN {X 0.129,Y -537.617,Z 1050.767,A 0.000,B 0.000,C 90.000,E1 353.970} C_DIS
LIN {X -0.099,Y -542.809,Z 1050.764,A 0.000,B 0.000,C 90.000,E1 353.451} C_DIS
LIN {X -0.265,Y -546.499,Z 1050.761,A 0.000,B 0.000,C 90.000,E1 353.053} C_DIS
LIN {X -0.076,Y -551.072,Z 1050.758,A 0.000,B 0.000,C 90.000,E1 352.470} C_DIS
LIN {X 0.065,Y -556.134,Z 1050.754,A 0.000,B 0.000,C 90.000,E1 351.781} C_DIS
LIN {X -0.229,Y -559.886,Z 1050.751,A 0.000,B 0.000,C 90.000,E1 351.254} C_DIS
LIN {X -0.179,Y -564.163,Z 1050.747,A 0.000,B 0.000,C 90.000,E1 350.557} C_DIS
LIN {X 0.054,Y -567.287,Z 1050.744,A 0.000,B 0.000,C 90.000,E1 349.982} C_DIS
LIN {X 0.165,Y -570.889,Z 1050.741,A 0.000,B 0.000,C 90.000,E1 349.285} C_DIS
LIN {X 0.181,Y -574.971,Z 1050.736,A 0.000,B 0.000,C 90.000,E1 348.465} C_DIS
LIN {X 0.243,Y -578.684,Z 1050.732,A 0.000,B 0.000,C 90.000,E1 347.645} C_DIS
LIN {X -0.001,Y -583.304,Z 1050.726,A 0.000,B 0.000,C 90.000,E1 346.589} C_DIS
LIN {X 0.280,Y -586.524,Z 1050.721,A 0.000,B 0.000,C 90.000,E1 345.755} C_DIS
LIN {X -0.023,Y -591.699,Z 1050.714,A 0.000,B 0.000,C 90.000,E1 344.448} C_DIS
LIN {X -0.244,Y -596.641,Z 1050.706,A 0.000,B 0.000,C 90.000,E1 343.142} C_DIS
LIN {X 0.076,Y -600.272,Z 1050.700,A 0.000,B 0.000,C 90.000,E1 342.054} C_DIS
LIN {X -0.314,Y -603.663,Z 1050.695,A 0.000,B 0.000,C 90.000,E1 341.040} C_DIS
LIN {X 0.306,Y -606.793,Z 1050.689,A 0.000,B 0.000,C 90.000,E1 339.934} C_DIS
LIN {X 0.142,Y -610.428,Z 1050.682,A 0.000,B 0.000,C 90.000,E1 338.646} C_DIS
LIN {X 0.031,Y -613.639,Z 1050.674,A 0.000,B 0.000,C 90.000,E1 337.358} C_DIS
LIN {X 0.228,Y -616.032,Z 1050.669,A 0.000,B 0.000,C 90.000,E1 336.305} C_DIS
LIN {X 0.164,Y -617.665,Z 1050.664,A 0.000,B 0.000,C 90.000,E1 335.537} C_DIS
LIN {X -0.141,Y -619.135,Z 1050.660,A 0.000,B 0.000,C 90.000,E1 334.793} C_DIS
LIN {X -0.175,Y -620.860,Z 1050.654,A 0.000,B 0.000,C 90.000,E1 333.768} C_DIS
LIN {X -0.183,Y -622.042,Z 1050.650,A 0.000,B 0.000,C 90.000,E1 332.999} C_DIS
LIN {X 0.117,Y -623.875,Z 1050.643,A 0.000,B 0.000,C 90.000,E1 331.691} C_DIS
LIN {X 0.147,Y -625.423,Z 1050.636,A 0.000,B 0.000,C 90.000,E1 330.411} C_DIS
LIN {X -0.053,Y -626.359,Z 1050.630,A 0.000,B 0.000,C 90.000,E1 329.410} C_DIS
LIN {X 0.097,Y -627.346,Z 1050.623,A 0.000,B 0.000,C 90.000,E1 328.122} C_DIS
LIN {X 0.266,Y -627.974,Z 1050.616,A 0.000,B 0.000,C 90.000,E1 326.834} C_DIS
LIN {X -0.080,Y -628.146,Z 1050.610,A 0.000,B 0.000,C 90.000,E1 325.849} C_DIS
LIN {X 0.089,Y -628.185,Z 1050.603,A 0.000,B 0.000,C 90.000,E1 324.562} C_DIS
LIN {X 0.093,Y -628.049,Z 1050.596,A 0.000,B 0.000,C 90.000,E1 323.290} C_DIS
LIN {X 0.012,Y -627.854,Z 1050.583,A 0.000,B 0.000,C 90.000,E1 321.009} C_DIS
LIN {X 0.124,Y -627.814,Z 1050.574,A 0.000,B 0.000,C 90.000,E1 319.218} C_DIS
LIN {X -0.334,Y -627.723,Z 1050.568,A 0.000,B 0.000,C 90.000,E1 318.243} C_DIS
LIN {X -0.295,Y -627.663,Z 1050.558,A 0.000,B 0.000,C 90.000,E1 316.458} C_DIS
LIN {X 0.219,Y -627.676,Z 1050.554,A 0.000,B 0.000,C 90.000,E1 315.648} C_DIS
LIN {X 0.365,Y -627.649,Z 1050.545,A 0.000,B 0.000,C 90.000,E1 314.109} C_DIS
LIN {X 0.070,Y -627.552,Z 1050.537,A 0.000,B 0.000,C 90.000,E1 312.609} C_DIS
LIN {X 0.153,Y -627.525,Z 1050.533,A 0.000,B 0.000,C 90.000,E1 311.838} C_DIS
LIN {X 0.117,Y -627.177,Z 1050.521,A 0.000,B 0.000,C 90.000,E1 309.806} C_DIS
LIN {X -0.348,Y -626.976,Z 1050.516,A 0.000,B 0.000,C 90.000,E1 308.830} C_DIS
LIN {X -0.132,Y -626.822,Z 1050.507,A 0.000,B 0.000,C 90.000,E1 307.282} C_DIS
LIN {X 0.032,Y -626.857,Z 1050.503,A 0.000,B 0.000,C 90.000,E1 306.503} C_DIS
LIN {X 0.199,Y -626.763,Z 1050.499,A 0.000,B 0.000,C 90.000,E1 305.724} C_DIS
LIN {X -0.195,Y -627.184,Z 1050.484,A 0.000,B 0.000,C 90.000,E1 303.214} C_DIS
LIN {X -0.019,Y -627.778,Z 1050.475,A 0.000,B 0.000,C 90.000,E1 301.416} C_DIS
LIN {X -0.339,Y -628.805,Z 1050.463,A 0.000,B 0.000,C 90.000,E1 299.411} C_DIS
LIN {X 0.104,Y -629.641,Z 1050.455,A 0.000,B 0.000,C 90.000,E1 297.847} C_DIS
LIN {X 0.130,Y -629.801,Z 1050.453,A 0.000,B 0.000,C 90.000,E1 297.590} C_DIS
LIN {X -0.292,Y -630.052,Z 1050.446,A 0.000,B 0.000,C 90.000,E1 296.360} C_DIS
LIN {X -0.182,Y -630.036,Z 1050.441,A 0.000,B 0.000,C 90.000,E1 295.335} C_DIS
LIN {X -0.130,Y -629.833,Z 1050.438,A 0.000,B 0.000,C 90.000,E1 294.823} C_DIS
LIN {X 0.284,Y -629.495,Z 1050.432,A 0.000,B 0.000,C 90.000,E1 293.770} C_DIS
LIN {X 0.120,Y -628.420,Z 1050.427,A 0.000,B 0.000,C 90.000,E1 292.770} C_DIS
LIN {X -0.086,Y -627.996,Z 1050.424,A 0.000,B 0.000,C 90.000,E1 292.280} C_DIS
LIN {X -0.072,Y -627.710,Z 1050.422,A 0.000,B 0.000,C 90.000,E1 292.025} C_DIS
LIN {X -0.283,Y -626.797,Z 1050.420,A 0.000,B 0.000,C 90.000,E1 291.535} C_DIS
LIN {X -0.274,Y -626.138,Z 1050.418,A 0.000,B 0.000,C 90.000,E1 291.280} C_DIS
LIN {X 0.313,Y -625.336,Z 1050.417,A 0.000,B 0.000,C 90.000,E1 290.972} C_DIS
LIN {X 0.091,Y -624.387,Z 1050.415,A 0.000,B 0.000,C 90.000,E1 290.737} C_DIS
LIN {X -0.139,Y -621.551,Z 1050.412,A 0.000,B 0.000,C 90.000,E1 290.248} C_DIS
LIN {X 0.195,Y -617.451,Z 1050.410,A 0.000,B 0.000,C 90.000,E1 289.704} C_DIS
LIN {X 0.180,Y -616.011,Z 1050.409,A 0.000,B 0.000,C 90.000,E1 289.577} C_DIS
LIN {X -0.182,Y -611.220,Z 1050.407,A 0.000,B 0.000,C 90.000,E1 289.268} C_DIS
LIN {X 0.081,Y -609.697,Z 1050.406,A 0.000,B 0.000,C 90.000,E1 289.141} C_DIS
LIN {X 0.044,Y -602.823,Z 1050.404,A 0.000,B 0.000,C 90.000,E1 288.779} C_DIS
LIN {X -0.268,Y -601.221,Z 1050.404,A 0.000,B 0.000,C 90.000,E1 288.725} C_DIS
LIN {X 0.091,Y -592.197,Z 1050.402,A 0.000,B 0.000,C 90.000,E1 288.308} C_DIS
LIN {X -0.162,Y -580.904,Z 1050.400,A 0.000,B 0.000,C 90.000,E1 288.000} C_DIS
LIN {X 0.021,Y -563.291,Z 1050.397,A 0.000,B 0.000,C 90.000,E1 287.511} C_DIS
LIN {X 0.189,Y -554.665,Z 1050.396,A 0.000,B 0.000,C 90.000,E1 287.275} C_DIS
LIN {X 0.121,Y -550.721,Z 1050.396,A 0.000,B 0.000,C 90.000,E1 287.166} C_DIS
LIN {X 0.253,Y -548.174,Z 1050.394,A 0.000,B 0.000,C 90.000,E1 286.913} C_DIS
LIN {X -0.145,Y -547.727,Z 1050.394,A 0.000,B 0.000,C 90.000,E1 286.858} C_DIS
LIN {X 0.102,Y -547.167,Z 1050.392,A 0.000,B 0.000,C 90.000,E1 286.551} C_DIS
LIN {X 0.093,Y -546.401,Z 1050.388,A 0.000,B 0.000,C 90.000,E1 285.788} C_DIS
LIN {X 0.074,Y -545.840,Z 1050.382,A 0.000,B 0.000,C 90.000,E1 284.662} C_DIS
LIN {X 0.047,Y -545.475,Z 1050.375,A 0.000,B 0.000,C 90.000,E1 283.536} C_DIS
LIN {X 0.097,Y -544.882,Z 1050.367,A 0.000,B 0.000,C 90.000,E1 282.119} C_DIS
LIN {X 0.011,Y -543.977,Z 1050.360,A 0.000,B 0.000,C 90.000,E1 280.715} C_DIS
LIN {X -0.108,Y -542.890,Z 1050.350,A 0.000,B 0.000,C 90.000,E1 279.029} C_DIS
LIN {X 0.128,Y -542.151,Z 1050.344,A 0.000,B 0.000,C 90.000,E1 277.871} C_DIS
LIN {X -0.176,Y -541.115,Z 1050.334,A 0.000,B 0.000,C 90.000,E1 276.201} C_DIS
LIN {X 0.030,Y -540.257,Z 1050.327,A 0.000,B 0.000,C 90.000,E1 274.759} C_DIS
LIN {X 0.203,Y -538.968,Z 1050.314,A 0.000,B 0.000,C 90.000,E1 272.465} C_DIS
LIN {X -0.225,Y -537.809,Z 1050.303,A 0.000,B 0.000,C 90.000,E1 270.516} C_DIS
LIN {X -0.163,Y -536.734,Z 1050.293,A 0.000,B 0.000,C 90.000,E1 268.797} C_DIS
LIN {X -0.119,Y -535.749,Z 1050.285,A 0.000,B 0.000,C 90.000,E1 267.364} C_DIS
LIN {X -0.059,Y -534.814,Z 1050.277,A 0.000,B 0.000,C 90.000,E1 265.927} C_DIS
LIN {X 0.012,Y -533.369,Z 1050.266,A 0.000,B 0.000,C 90.000,E1 263.913} C_DIS
LIN {X 0.007,Y -532.627,Z 1050.261,A 0.000,B 0.000,C 90.000,E1 263.053} C_DIS
LIN {X 0.091,Y -531.438,Z 1050.255,A 0.000,B 0.000,C 90.000,E1 261.894} C_DIS
LIN {X 0.268,Y -529.282,Z 1050.244,A 0.000,B 0.000,C 90.000,E1 259.859} C_DIS
LIN {X -0.219,Y -528.020,Z 1050.237,A 0.000,B 0.000,C 90.000,E1 258.757} C_DIS
LIN {X 0.028,Y -526.465,Z 1050.229,A 0.000,B 0.000,C 90.000,E1 257.285} C_DIS
LIN {X -0.214,Y -524.024,Z 1050.217,A 0.000,B 0.000,C 90.000,E1 254.991} C_DIS
LIN {X 0.238,Y -522.150,Z 1050.207,A 0.000,B 0.000,C 90.000,E1 253.196} C_DIS
LIN {X 0.006,Y -520.571,Z 1050.199,A 0.000,B 0.000,C 90.000,E1 251.764} C_DIS
LIN {X 0.072,Y -518.845,Z 1050.191,A 0.000,B 0.000,C 90.000,E1 250.296} C_DIS
LIN {X 0.066,Y -516.713,Z 1050.181,A 0.000,B 0.000,C 90.000,E1 248.539} C_DIS
LIN {X 0.120,Y -515.284,Z 1050.174,A 0.000,B 0.000,C 90.000,E1 247.358} C_DIS
LIN {X -0.074,Y -512.728,Z 1050.165,A 0.000,B 0.000,C 90.000,E1 245.613} C_DIS
LIN {X -0.221,Y -510.455,Z 1050.156,A 0.000,B 0.000,C 90.000,E1 244.152} C_DIS
LIN {X -0.180,Y -508.028,Z 1050.148,A 0.000,B 0.000,C 90.000,E1 242.666} C_DIS
LIN {X -0.181,Y -505.460,Z 1050.140,A 0.000,B 0.000,C 90.000,E1 241.179} C_DIS
LIN {X 0.135,Y -503.329,Z 1050.133,A 0.000,B 0.000,C 90.000,E1 239.950} C_DIS
LIN {X 0.004,Y -499.445,Z 1050.122,A 0.000,B 0.000,C 90.000,E1 237.867} C_DIS
LIN {X 0.312,Y -497.174,Z 1050.115,A 0.000,B 0.000,C 90.000,E1 236.628} C_DIS
LIN {X -0.102,Y -494.769,Z 1050.108,A 0.000,B 0.000,C 90.000,E1 235.468} C_DIS
LIN {X -0.273,Y -492.286,Z 1050.101,A 0.000,B 0.000,C 90.000,E1 234.276} C_DIS
LIN {X 0.181,Y -488.095,Z 1050.091,A 0.000,B 0.000,C 90.000,E1 232.396} C_DIS
LIN {X -0.018,Y -483.108,Z 1050.079,A 0.000,B 0.000,C 90.000,E1 230.275} C_DIS
LIN {X 0.030,Y -479.713,Z 1050.071,A 0.000,B 0.000,C 90.000,E1 228.728} C_DIS
LIN {X -0.039,Y -476.548,Z 1050.062,A 0.000,B 0.000,C 90.000,E1 227.187} C_DIS
LIN {X 0.106,Y -471.462,Z 1050.048,A 0.000,B 0.000,C 90.000,E1 224.676} C_DIS
LIN {X -0.130,Y -468.323,Z 1050.040,A 0.000,B 0.000,C 90.000,E1 223.137} C_DIS
LIN {X 0.061,Y -463.868,Z 1050.027,A 0.000,B 0.000,C 90.000,E1 220.906} C_DIS
LIN {X 0.044,Y -460.519,Z 1050.019,A 0.000,B 0.000,C 90.000,E1 219.322} C_DIS
LIN {X -0.041,Y -454.496,Z 1050.003,A 0.000,B 0.000,C 90.000,E1 216.457} C_DIS
LIN {X -0.007,Y -449.843,Z 1049.990,A 0.000,B 0.000,C 90.000,E1 214.199} C_DIS
LIN {X 0.248,Y -446.536,Z 1049.981,A 0.000,B 0.000,C 90.000,E1 212.546} C_DIS
LIN {X 0.192,Y -442.984,Z 1049.972,A 0.000,B 0.000,C 90.000,E1 210.924} C_DIS
LIN {X -0.120,Y -438.608,Z 1049.961,A 0.000,B 0.000,C 90.000,E1 208.999} C_DIS
LIN {X 0.025,Y -434.364,Z 1049.950,A 0.000,B 0.000,C 90.000,E1 207.001} C_DIS
LIN {X -0.135,Y -432.300,Z 1049.945,A 0.000,B 0.000,C 90.000,E1 206.027} C_DIS
LIN {X 0.211,Y -425.535,Z 1049.926,A 0.000,B 0.000,C 90.000,E1 202.642} C_DIS
LIN {X -0.015,Y -419.393,Z 1049.905,A 0.000,B 0.000,C 90.000,E1 198.960} C_DIS
LIN {X 0.122,Y -417.612,Z 1049.898,A 0.000,B 0.000,C 90.000,E1 197.583} C_DIS
LIN {X 0.080,Y -416.648,Z 1049.892,A 0.000,B 0.000,C 90.000,E1 196.567} C_DIS
LIN {X -0.012,Y -416.132,Z 1049.888,A 0.000,B 0.000,C 90.000,E1 195.898} C_DIS
LIN {X 0.176,Y -415.808,Z 1049.885,A 0.000,B 0.000,C 90.000,E1 195.190} C_DIS
LIN {X -0.038,Y -415.519,Z 1049.881,A 0.000,B 0.000,C 90.000,E1 194.537} C_DIS
LIN {X 0.146,Y -415.703,Z 1049.877,A 0.000,B 0.000,C 90.000,E1 193.828} C_DIS
LIN {X -0.073,Y -416.304,Z 1049.873,A 0.000,B 0.000,C 90.000,E1 193.175} C_DIS
LIN {X 0.024,Y -417.389,Z 1049.869,A 0.000,B 0.000,C 90.000,E1 192.479} C_DIS
LIN {X -0.189,Y -419.269,Z 1049.866,A 0.000,B 0.000,C 90.000,E1 191.827} C_DIS
LIN {X -0.056,Y -421.243,Z 1049.863,A 0.000,B 0.000,C 90.000,E1 191.299} C_DIS
LIN {X 0.090,Y -424.561,Z 1049.859,A 0.000,B 0.000,C 90.000,E1 190.602} C_DIS
LIN {X -0.155,Y -428.358,Z 1049.855,A 0.000,B 0.000,C 90.000,E1 189.962} C_DIS
LIN {X 0.186,Y -442.371,Z 1049.843,A 0.000,B 0.000,C 90.000,E1 187.757} C_DIS
LIN {X -0.002,Y -452.626,Z 1049.835,A 0.000,B 0.000,C 90.000,E1 186.315} C_DIS
LIN {X -0.061,Y -462.731,Z 1049.827,A 0.000,B 0.000,C 90.000,E1 184.878} C_DIS
LIN {X -0.177,Y -470.105,Z 1049.821,A 0.000,B 0.000,C 90.000,E1 183.784} C_DIS
LIN {X 0.113,Y -476.196,Z 1049.816,A 0.000,B 0.000,C 90.000,E1 182.808} C_DIS
LIN {X -0.194,Y -484.020,Z 1049.809,A 0.000,B 0.000,C 90.000,E1 181.604} C_DIS
LIN {X 0.087,Y -488.739,Z 1049.805,A 0.000,B 0.000,C 90.000,E1 180.802} C_DIS
LIN {X -0.046,Y -496.136,Z 1049.798,A 0.000,B 0.000,C 90.000,E1 179.599} C_DIS
LIN {X -0.137,Y -500.612,Z 1049.794,A 0.000,B 0.000,C 90.000,E1 178.854} C_DIS
LIN {X 0.116,Y -508.436,Z 1049.786,A 0.000,B 0.000,C 90.000,E1 177.478} C_DIS
LIN {X -0.139,Y -513.498,Z 1049.781,A 0.000,B 0.000,C 90.000,E1 176.617} C_DIS
LIN {X 0.027,Y -523.421,Z 1049.771,A 0.000,B 0.000,C 90.000,E1 174.837} C_DIS
LIN {X 0.185,Y -530.697,Z 1049.764,A 0.000,B 0.000,C 90.000,E1 173.514} C_DIS
LIN {X -0.058,Y -536.209,Z 1049.759,A 0.000,B 0.000,C 90.000,E1 172.534} C_DIS
LIN {X 0.181,Y -544.043,Z 1049.751,A 0.000,B 0.000,C 90.000,E1 171.084} C_DIS
LIN {X -0.137,Y -552.380,Z 1049.742,A 0.000,B 0.000,C 90.000,E1 169.567} C_DIS
LIN {X -0.025,Y -557.607,Z 1049.737,A 0.000,B 0.000,C 90.000,E1 168.578} C_DIS
LIN {X 0.147,Y -562.638,Z 1049.731,A 0.000,B 0.000,C 90.000,E1 167.589} C_DIS
LIN {X -0.052,Y -567.638,Z 1049.726,A 0.000,B 0.000,C 90.000,E1 166.645} C_DIS
LIN {X -0.187,Y -572.368,Z 1049.720,A 0.000,B 0.000,C 90.000,E1 165.700} C_DIS
LIN {X 0.188,Y -577.600,Z 1049.714,A 0.000,B 0.000,C 90.000,E1 164.574} C_DIS
LIN {X 0.168,Y -582.027,Z 1049.709,A 0.000,B 0.000,C 90.000,E1 163.630} C_DIS
LIN {X 0.283,Y -586.797,Z 1049.703,A 0.000,B 0.000,C 90.000,E1 162.543} C_DIS
LIN {X 0.044,Y -590.211,Z 1049.699,A 0.000,B 0.000,C 90.000,E1 161.764} C_DIS
LIN {X -0.290,Y -594.434,Z 1049.693,A 0.000,B 0.000,C 90.000,E1 160.732} C_DIS
LIN {X -0.104,Y -599.457,Z 1049.686,A 0.000,B 0.000,C 90.000,E1 159.390} C_DIS
LIN {X -0.098,Y -603.187,Z 1049.680,A 0.000,B 0.000,C 90.000,E1 158.337} C_DIS
LIN {X 0.025,Y -605.867,Z 1049.675,A 0.000,B 0.000,C 90.000,E1 157.539} C_DIS
LIN {X 0.071,Y -609.928,Z 1049.668,A 0.000,B 0.000,C 90.000,E1 156.230} C_DIS
LIN {X 0.180,Y -613.731,Z 1049.661,A 0.000,B 0.000,C 90.000,E1 154.921} C_DIS
LIN {X 0.098,Y -615.892,Z 1049.656,A 0.000,B 0.000,C 90.000,E1 154.152} C_DIS
LIN {X 0.024,Y -618.626,Z 1049.651,A 0.000,B 0.000,C 90.000,E1 153.127} C_DIS
LIN {X -0.021,Y -621.884,Z 1049.644,A 0.000,B 0.000,C 90.000,E1 151.847} C_DIS
LIN {X 0.273,Y -623.802,Z 1049.639,A 0.000,B 0.000,C 90.000,E1 151.051} C_DIS
LIN {X 0.076,Y -627.570,Z 1049.631,A 0.000,B 0.000,C 90.000,E1 149.537} C_DIS
LIN {X 0.271,Y -631.015,Z 1049.622,A 0.000,B 0.000,C 90.000,E1 147.995} C_DIS
LIN {X 0.146,Y -633.313,Z 1049.617,A 0.000,B 0.000,C 90.000,E1 146.993} C_DIS
LIN {X -0.116,Y -636.102,Z 1049.610,A 0.000,B 0.000,C 90.000,E1 145.754} C_DIS
LIN {X -0.094,Y -639.410,Z 1049.601,A 0.000,B 0.000,C 90.000,E1 144.242} C_DIS
LIN {X 0.141,Y -642.730,Z 1049.593,A 0.000,B 0.000,C 90.000,E1 142.718} C_DIS
LIN {X -0.205,Y -646.067,Z 1049.585,A 0.000,B 0.000,C 90.000,E1 141.251} C_DIS
LIN {X -0.070,Y -649.329,Z 1049.576,A 0.000,B 0.000,C 90.000,E1 139.747} C_DIS
LIN {X 0.134,Y -652.616,Z 1049.568,A 0.000,B 0.000,C 90.000,E1 138.243} C_DIS
LIN {X -0.168,Y -657.122,Z 1049.557,A 0.000,B 0.000,C 90.000,E1 136.296} C_DIS
LIN {X 0.067,Y -664.077,Z 1049.542,A 0.000,B 0.000,C 90.000,E1 133.581} C_DIS
LIN {X 0.030,Y -668.731,Z 1049.533,A 0.000,B 0.000,C 90.000,E1 131.881} C_DIS
LIN {X 0.195,Y -673.347,Z 1049.523,A 0.000,B 0.000,C 90.000,E1 130.172} C_DIS
LIN {X -0.065,Y -677.244,Z 1049.515,A 0.000,B 0.000,C 90.000,E1 128.749} C_DIS
LIN {X -0.144,Y -681.007,Z 1049.507,A 0.000,B 0.000,C 90.000,E1 127.317} C_DIS
LIN {X -0.125,Y -685.240,Z 1049.498,A 0.000,B 0.000,C 90.000,E1 125.644} C_DIS
LIN {X -0.091,Y -688.247,Z 1049.491,A 0.000,B 0.000,C 90.000,E1 124.452} C_DIS
LIN {X -0.177,Y -691.800,Z 1049.484,A 0.000,B 0.000,C 90.000,E1 123.038} C_DIS
LIN {X -0.414,Y -694.598,Z 1049.477,A 0.000,B 0.000,C 90.000,E1 121.878} C_DIS
LIN {X -0.271,Y -696.728,Z 1049.472,A 0.000,B 0.000,C 90.000,E1 120.924} C_DIS
LIN {X 0.143,Y -698.581,Z 1049.467,A 0.000,B 0.000,C 90.000,E1 119.951} C_DIS
LIN {X -0.282,Y -699.698,Z 1049.463,A 0.000,B 0.000,C 90.000,E1 119.283} C_DIS
LIN {X -0.090,Y -700.624,Z 1049.459,A 0.000,B 0.000,C 90.000,E1 118.565} C_DIS
LIN {X -0.029,Y -702.443,Z 1049.450,A 0.000,B 0.000,C 90.000,E1 116.924} C_DIS
LIN {X 0.149,Y -703.436,Z 1049.444,A 0.000,B 0.000,C 90.000,E1 115.976} C_DIS
LIN {X -0.010,Y -704.253,Z 1049.438,A 0.000,B 0.000,C 90.000,E1 114.823} C_DIS
LIN {X -0.021,Y -704.297,Z 1049.437,A 0.000,B 0.000,C 90.000,E1 114.591} C_DIS
LIN {X -0.093,Y -704.069,Z 1049.434,A 0.000,B 0.000,C 90.000,E1 114.131} C_DIS
LIN {X -0.097,Y -703.623,Z 1049.433,A 0.000,B 0.000,C 90.000,E1 113.898} C_DIS
LIN {X -0.180,Y -702.417,Z 1049.430,A 0.000,B 0.000,C 90.000,E1 113.439} C_DIS
LIN {X -0.321,Y -701.847,Z 1049.430,A 0.000,B 0.000,C 90.000,E1 113.334} C_DIS
LIN {X 0.222,Y -698.846,Z 1049.427,A 0.000,B 0.000,C 90.000,E1 112.823} C_DIS
LIN {X 0.084,Y -697.905,Z 1049.426,A 0.000,B 0.000,C 90.000,E1 112.717} C_DIS
LIN {X 0.214,Y -696.497,Z 1049.426,A 0.000,B 0.000,C 90.000,E1 112.589} C_DIS
LIN {X 0.236,Y -692.597,Z 1049.425,A 0.000,B 0.000,C 90.000,E1 112.386} C_DIS
LIN {X 0.199,Y -687.559,Z 1049.423,A 0.000,B 0.000,C 90.000,E1 112.153} C_DIS
LIN {X 0.226,Y -685.333,Z 1049.423,A 0.000,B 0.000,C 90.000,E1 112.078} C_DIS
LIN {X -0.205,Y -683.667,Z 1049.423,A 0.000,B 0.000,C 90.000,E1 112.078} C_DIS
LIN {X -0.116,Y -675.641,Z 1049.422,A 0.000,B 0.000,C 90.000,E1 111.972} C_DIS
LIN {X -0.152,Y -610.055,Z 1049.422,A 0.000,B 0.000,C 90.000,E1 111.972} C_DIS
LIN {X -0.218,Y -604.236,Z 1049.421,A 0.000,B 0.000,C 90.000,E1 111.770} C_DIS
LIN {X 0.156,Y -597.847,Z 1049.419,A 0.000,B 0.000,C 90.000,E1 111.408} C_DIS
LIN {X 0.161,Y -592.465,Z 1049.417,A 0.000,B 0.000,C 90.000,E1 111.046} C_DIS
LIN {X -0.032,Y -575.721,Z 1049.410,A 0.000,B 0.000,C 90.000,E1 109.704} C_DIS
LIN {X -0.193,Y -569.680,Z 1049.407,A 0.000,B 0.000,C 90.000,E1 109.268} C_DIS
LIN {X 0.264,Y -561.329,Z 1049.404,A 0.000,B 0.000,C 90.000,E1 108.725} C_DIS
LIN {X -0.221,Y -554.740,Z 1049.402,A 0.000,B 0.000,C 90.000,E1 108.417} C_DIS
LIN {X 0.084,Y -549.652,Z 1049.400,A 0.000,B 0.000,C 90.000,E1 108.055} C_DIS
LIN {X 0.232,Y -547.792,Z 1049.399,A 0.000,B 0.000,C 90.000,E1 107.819} C_DIS
LIN {X 0.190,Y -547.779,Z 1049.399,A 0.000,B 0.000,C 90.000,E1 107.819} C_DIS
LIN {X 0.275,Y -547.318,Z 1049.397,A 0.000,B 0.000,C 90.000,E1 107.511} C_DIS
LIN {X 0.124,Y -548.647,Z 1049.384,A 0.000,B 0.000,C 90.000,E1 105.134} C_DIS
LIN {X -0.159,Y -550.596,Z 1049.369,A 0.000,B 0.000,C 90.000,E1 102.355} C_DIS
LIN {X -0.065,Y -553.565,Z 1049.351,A 0.000,B 0.000,C 90.000,E1 99.265} C_DIS
LIN {X 0.084,Y -555.753,Z 1049.341,A 0.000,B 0.000,C 90.000,E1 97.296} C_DIS
LIN {X -0.102,Y -557.068,Z 1049.334,A 0.000,B 0.000,C 90.000,E1 96.201} C_DIS
LIN {X -0.269,Y -558.200,Z 1049.328,A 0.000,B 0.000,C 90.000,E1 95.106} C_DIS
LIN {X 0.129,Y -559.119,Z 1049.322,A 0.000,B 0.000,C 90.000,E1 93.955} C_DIS
LIN {X 0.030,Y -559.951,Z 1049.314,A 0.000,B 0.000,C 90.000,E1 92.579} C_DIS
LIN {X -0.237,Y -560.346,Z 1049.310,A 0.000,B 0.000,C 90.000,E1 91.776} C_DIS
LIN {X -0.235,Y -560.995,Z 1049.301,A 0.000,B 0.000,C 90.000,E1 90.115} C_DIS
LIN {X 0.248,Y -561.426,Z 1049.293,A 0.000,B 0.000,C 90.000,E1 88.682} C_DIS
LIN {X -0.276,Y -561.949,Z 1049.284,A 0.000,B 0.000,C 90.000,E1 87.078} C_DIS
LIN {X 0.270,Y -562.487,Z 1049.276,A 0.000,B 0.000,C 90.000,E1 85.641} C_DIS
LIN {X 0.269,Y -562.887,Z 1049.268,A 0.000,B 0.000,C 90.000,E1 84.261} C_DIS
LIN {X -0.226,Y -563.247,Z 1049.261,A 0.000,B 0.000,C 90.000,E1 82.932} C_DIS
LIN {X 0.238,Y -563.885,Z 1049.248,A 0.000,B 0.000,C 90.000,E1 80.679} C_DIS
LIN {X -0.053,Y -564.873,Z 1049.235,A 0.000,B 0.000,C 90.000,E1 78.229} C_DIS
LIN {X 0.229,Y -565.591,Z 1049.227,A 0.000,B 0.000,C 90.000,E1 76.825} C_DIS
LIN {X 0.204,Y -566.918,Z 1049.215,A 0.000,B 0.000,C 90.000,E1 74.629} C_DIS
LIN {X -0.115,Y -568.180,Z 1049.206,A 0.000,B 0.000,C 90.000,E1 73.015} C_DIS
LIN {X 0.272,Y -570.000,Z 1049.193,A 0.000,B 0.000,C 90.000,E1 70.786} C_DIS
LIN {X 0.027,Y -571.113,Z 1049.186,A 0.000,B 0.000,C 90.000,E1 69.444} C_DIS
LIN {X 0.150,Y -572.298,Z 1049.177,A 0.000,B 0.000,C 90.000,E1 67.794} C_DIS
LIN {X -0.189,Y -573.574,Z 1049.166,A 0.000,B 0.000,C 90.000,E1 65.921} C_DIS
LIN {X -0.104,Y -574.520,Z 1049.157,A 0.000,B 0.000,C 90.000,E1 64.280} C_DIS
LIN {X 0.248,Y -575.332,Z 1049.148,A 0.000,B 0.000,C 90.000,E1 62.615} C_DIS
LIN {X 0.101,Y -576.099,Z 1049.139,A 0.000,B 0.000,C 90.000,E1 61.001} C_DIS
LIN {X -0.257,Y -576.878,Z 1049.130,A 0.000,B 0.000,C 90.000,E1 59.410} C_DIS
LIN {X -0.128,Y -577.221,Z 1049.125,A 0.000,B 0.000,C 90.000,E1 58.584} C_DIS
LIN {X -0.307,Y -577.706,Z 1049.118,A 0.000,B 0.000,C 90.000,E1 57.248} C_DIS
LIN {X -0.015,Y -578.142,Z 1049.109,A 0.000,B 0.000,C 90.000,E1 55.595} C_DIS
LIN {X -0.016,Y -578.478,Z 1049.101,A 0.000,B 0.000,C 90.000,E1 54.242} C_DIS
LIN {X 0.131,Y -578.563,Z 1049.097,A 0.000,B 0.000,C 90.000,E1 53.417} C_DIS
LIN {X -0.030,Y -578.508,Z 1049.091,A 0.000,B 0.000,C 90.000,E1 52.351} C_DIS
LIN {X 0.159,Y -578.288,Z 1049.085,A 0.000,B 0.000,C 90.000,E1 51.251} C_DIS
LIN {X 0.187,Y -578.010,Z 1049.080,A 0.000,B 0.000,C 90.000,E1 50.436} C_DIS
LIN {X 0.078,Y -577.400,Z 1049.073,A 0.000,B 0.000,C 90.000,E1 49.094} C_DIS
LIN {X 0.189,Y -576.786,Z 1049.067,A 0.000,B 0.000,C 90.000,E1 48.000} C_DIS
LIN {X 0.147,Y -575.599,Z 1049.058,A 0.000,B 0.000,C 90.000,E1 46.377} C_DIS
LIN {X -0.180,Y -574.421,Z 1049.052,A 0.000,B 0.000,C 90.000,E1 45.324} C_DIS
LIN {X 0.059,Y -573.782,Z 1049.049,A 0.000,B 0.000,C 90.000,E1 44.757} C_DIS
LIN {X 0.221,Y -571.764,Z 1049.041,A 0.000,B 0.000,C 90.000,E1 43.380} C_DIS
LIN {X 0.251,Y -569.900,Z 1049.035,A 0.000,B 0.000,C 90.000,E1 42.285} C_DIS
LIN {X 0.183,Y -568.354,Z 1049.031,A 0.000,B 0.000,C 90.000,E1 41.472} C_DIS
LIN {X 0.162,Y -566.013,Z 1049.024,A 0.000,B 0.000,C 90.000,E1 40.378} C_DIS
LIN {X -0.165,Y -562.402,Z 1049.017,A 0.000,B 0.000,C 90.000,E1 39.036} C_DIS
LIN {X 0.231,Y -558.881,Z 1049.011,A 0.000,B 0.000,C 90.000,E1 37.890} C_DIS
LIN {X -0.031,Y -556.984,Z 1049.008,A 0.000,B 0.000,C 90.000,E1 37.363} C_DIS
LIN {X 0.134,Y -554.899,Z 1049.005,A 0.000,B 0.000,C 90.000,E1 36.790} C_DIS
LIN {X 0.029,Y -551.456,Z 1049.000,A 0.000,B 0.000,C 90.000,E1 35.964} C_DIS
LIN {X 0.211,Y -547.810,Z 1048.995,A 0.000,B 0.000,C 90.000,E1 35.105} C_DIS
LIN {X 0.167,Y -544.432,Z 1048.991,A 0.000,B 0.000,C 90.000,E1 34.405} C_DIS
LIN {X 0.092,Y -540.787,Z 1048.987,A 0.000,B 0.000,C 90.000,E1 33.706} C_DIS
LIN {X -0.305,Y -535.394,Z 1048.982,A 0.000,B 0.000,C 90.000,E1 32.752} C_DIS
LIN {X -0.022,Y -529.550,Z 1048.976,A 0.000,B 0.000,C 90.000,E1 31.720} C_DIS
LIN {X 0.049,Y -524.040,Z 1048.971,A 0.000,B 0.000,C 90.000,E1 30.846} C_DIS
LIN {X 0.123,Y -520.101,Z 1048.968,A 0.000,B 0.000,C 90.000,E1 30.256} C_DIS
LIN {X 0.079,Y -516.991,Z 1048.966,A 0.000,B 0.000,C 90.000,E1 29.823} C_DIS
LIN {X -0.089,Y -512.620,Z 1048.963,A 0.000,B 0.000,C 90.000,E1 29.255} C_DIS
LIN {X -0.009,Y -505.452,Z 1048.958,A 0.000,B 0.000,C 90.000,E1 28.359} C_DIS
LIN {X -0.036,Y -500.253,Z 1048.954,A 0.000,B 0.000,C 90.000,E1 27.769} C_DIS
LIN {X 0.045,Y -493.619,Z 1048.950,A 0.000,B 0.000,C 90.000,E1 27.052} C_DIS
LIN {X -0.255,Y -483.969,Z 1048.945,A 0.000,B 0.000,C 90.000,E1 26.104} C_DIS
LIN {X 0.026,Y -472.540,Z 1048.939,A 0.000,B 0.000,C 90.000,E1 24.975} C_DIS
LIN {X 0.082,Y -462.074,Z 1048.934,A 0.000,B 0.000,C 90.000,E1 24.027} C_DIS
LIN {X -0.181,Y -449.840,Z 1048.928,A 0.000,B 0.000,C 90.000,E1 23.025} C_DIS
LIN {X 0.086,Y -427.361,Z 1048.917,A 0.000,B 0.000,C 90.000,E1 20.972} C_DIS
LIN {X -0.093,Y -417.397,Z 1048.911,A 0.000,B 0.000,C 90.000,E1 19.993} C_DIS
LIN {X -0.027,Y -407.585,Z 1048.905,A 0.000,B 0.000,C 90.000,E1 18.906} C_DIS
LIN {X -0.174,Y -399.575,Z 1048.900,A 0.000,B 0.000,C 90.000,E1 17.946} C_DIS
LIN {X 0.150,Y -395.299,Z 1048.896,A 0.000,B 0.000,C 90.000,E1 17.275} C_DIS
LIN {X -0.139,Y -393.169,Z 1048.894,A 0.000,B 0.000,C 90.000,E1 16.858} C_DIS
LIN {X -0.055,Y -391.814,Z 1048.891,A 0.000,B 0.000,C 90.000,E1 16.315} C_DIS
LIN {X -0.110,Y -391.499,Z 1048.887,A 0.000,B 0.000,C 90.000,E1 15.607} C_DIS
LIN {X -0.096,Y -391.857,Z 1048.883,A 0.000,B 0.000,C 90.000,E1 14.898} C_DIS
LIN {X 0.178,Y -398.376,Z 1048.855,A 0.000,B 0.000,C 90.000,E1 9.905} C_DIS
LIN {X -0.039,Y -405.547,Z 1048.834,A 0.000,B 0.000,C 90.000,E1 6.087} C_DIS
LIN {X -0.084,Y -409.333,Z 1048.824,A 0.000,B 0.000,C 90.000,E1 4.359} C_DIS
LIN {X -0.099,Y -411.857,Z 1048.818,A 0.000,B 0.000,C 90.000,E1 3.326} C_DIS
LIN {X 0.076,Y -414.225,Z 1048.815,A 0.000,B 0.000,C 90.000,E1 2.751} C_DIS
LIN {X 0.082,Y -416.354,Z 1048.813,A 0.000,B 0.000,C 90.000,E1 2.407} C_DIS
LIN {X 0.088,Y -417.508,Z 1048.813,A 0.000,B 0.000,C 90.000,E1 2.236} C_DIS
LIN {X -0.169,Y -422.105,Z 1048.810,A 0.000,B 0.000,C 90.000,E1 1.833} C_DIS
LIN {X 0.106,Y -431.411,Z 1048.807,A 0.000,B 0.000,C 90.000,E1 1.203} C_DIS
LIN {X 0.086,Y -452.256,Z 1048.799,A 0.000,B 0.000,C 90.000,E1 359.885} C_DIS
LIN {X 0.142,Y -473.748,Z 1048.792,A 0.000,B 0.000,C 90.000,E1 358.568} C_DIS
LIN {X -0.076,Y -488.307,Z 1048.787,A 0.000,B 0.000,C 90.000,E1 357.707} C_DIS
LIN {X 0.134,Y -497.857,Z 1048.784,A 0.000,B 0.000,C 90.000,E1 357.078} C_DIS
LIN {X 0.107,Y -505.622,Z 1048.781,A 0.000,B 0.000,C 90.000,E1 356.560} C_DIS
LIN {X -0.164,Y -511.750,Z 1048.779,A 0.000,B 0.000,C 90.000,E1 356.159} C_DIS
LIN {X -0.068,Y -517.852,Z 1048.776,A 0.000,B 0.000,C 90.000,E1 355.698} C_DIS
LIN {X -0.195,Y -525.131,Z 1048.773,A 0.000,B 0.000,C 90.000,E1 355.122} C_DIS
LIN {X -0.193,Y -533.513,Z 1048.769,A 0.000,B 0.000,C 90.000,E1 354.375} C_DIS
LIN {X 0.108,Y -540.111,Z 1048.765,A 0.000,B 0.000,C 90.000,E1 353.685} C_DIS
LIN {X -0.181,Y -545.231,Z 1048.762,A 0.000,B 0.000,C 90.000,E1 353.166} C_DIS
LIN {X -0.025,Y -549.873,Z 1048.759,A 0.000,B 0.000,C 90.000,E1 352.591} C_DIS
LIN {X -0.250,Y -555.050,Z 1048.755,A 0.000,B 0.000,C 90.000,E1 351.951} C_DIS
LIN {X -0.198,Y -559.775,Z 1048.751,A 0.000,B 0.000,C 90.000,E1 351.254} C_DIS
LIN {X -0.149,Y -564.080,Z 1048.748,A 0.000,B 0.000,C 90.000,E1 350.557} C_DIS
LIN {X -0.061,Y -567.986,Z 1048.744,A 0.000,B 0.000,C 90.000,E1 349.859} C_DIS
LIN {X -0.180,Y -572.284,Z 1048.739,A 0.000,B 0.000,C 90.000,E1 349.050} C_DIS
LIN {X -0.150,Y -576.308,Z 1048.735,A 0.000,B 0.000,C 90.000,E1 348.229} C_DIS
LIN {X -0.075,Y -579.934,Z 1048.730,A 0.000,B 0.000,C 90.000,E1 347.409} C_DIS
LIN {X 0.031,Y -583.411,Z 1048.726,A 0.000,B 0.000,C 90.000,E1 346.589} C_DIS
LIN {X 0.313,Y -586.652,Z 1048.721,A 0.000,B 0.000,C 90.000,E1 345.755} C_DIS
LIN {X 0.013,Y -591.859,Z 1048.714,A 0.000,B 0.000,C 90.000,E1 344.448} C_DIS
LIN {X -0.205,Y -596.835,Z 1048.706,A 0.000,B 0.000,C 90.000,E1 343.142} C_DIS
LIN {X 0.118,Y -600.487,Z 1048.700,A 0.000,B 0.000,C 90.000,E1 342.054} C_DIS
LIN {X -0.269,Y -603.934,Z 1048.695,A 0.000,B 0.000,C 90.000,E1 341.040} C_DIS
LIN {X 0.355,Y -607.055,Z 1048.689,A 0.000,B 0.000,C 90.000,E1 339.934} C_DIS
LIN {X -0.262,Y -609.258,Z 1048.684,A 0.000,B 0.000,C 90.000,E1 339.209} C_DIS
LIN {X 0.197,Y -610.724,Z 1048.682,A 0.000,B 0.000,C 90.000,E1 338.646} C_DIS
LIN {X 0.090,Y -613.971,Z 1048.674,A 0.000,B 0.000,C 90.000,E1 337.358} C_DIS
LIN {X -0.271,Y -616.374,Z 1048.669,A 0.000,B 0.000,C 90.000,E1 336.357} C_DIS
LIN {X 0.232,Y -618.032,Z 1048.664,A 0.000,B 0.000,C 90.000,E1 335.537} C_DIS
LIN {X -0.079,Y -620.007,Z 1048.659,A 0.000,B 0.000,C 90.000,E1 334.537} C_DIS
LIN {X -0.100,Y -621.709,Z 1048.653,A 0.000,B 0.000,C 90.000,E1 333.512} C_DIS
LIN {X -0.098,Y -623.282,Z 1048.647,A 0.000,B 0.000,C 90.000,E1 332.487} C_DIS
LIN {X 0.216,Y -624.712,Z 1048.641,A 0.000,B 0.000,C 90.000,E1 331.435} C_DIS
LIN {X -0.296,Y -625.959,Z 1048.636,A 0.000,B 0.000,C 90.000,E1 330.461} C_DIS
LIN {X 0.062,Y -627.154,Z 1048.629,A 0.000,B 0.000,C 90.000,E1 329.154} C_DIS
LIN {X 0.214,Y -628.011,Z 1048.623,A 0.000,B 0.000,C 90.000,E1 328.122} C_DIS
LIN {X -0.126,Y -628.749,Z 1048.615,A 0.000,B 0.000,C 90.000,E1 326.628} C_DIS
LIN {X 0.057,Y -628.930,Z 1048.609,A 0.000,B 0.000,C 90.000,E1 325.595} C_DIS
LIN {X 0.240,Y -629.000,Z 1048.603,A 0.000,B 0.000,C 90.000,E1 324.562} C_DIS
LIN {X -0.245,Y -628.932,Z 1048.596,A 0.000,B 0.000,C 90.000,E1 323.336} C_DIS
LIN {X 0.205,Y -628.824,Z 1048.583,A 0.000,B 0.000,C 90.000,E1 321.009} C_DIS
LIN {X -0.200,Y -628.917,Z 1048.572,A 0.000,B 0.000,C 90.000,E1 319.013} C_DIS
LIN {X -0.040,Y -628.846,Z 1048.558,A 0.000,B 0.000,C 90.000,E1 316.458} C_DIS
LIN {X 0.367,Y -628.860,Z 1048.552,A 0.000,B 0.000,C 90.000,E1 315.405} C_DIS
LIN {X -0.232,Y -628.904,Z 1048.545,A 0.000,B 0.000,C 90.000,E1 314.190} C_DIS
LIN {X 0.141,Y -628.871,Z 1048.534,A 0.000,B 0.000,C 90.000,E1 312.123} C_DIS
LIN {X -0.059,Y -628.817,Z 1048.531,A 0.000,B 0.000,C 90.000,E1 311.634} C_DIS
LIN {X 0.351,Y -628.579,Z 1048.520,A 0.000,B 0.000,C 90.000,E1 309.564} C_DIS
LIN {X 0.251,Y -628.390,Z 1048.513,A 0.000,B 0.000,C 90.000,E1 308.302} C_DIS
LIN {X 0.089,Y -628.327,Z 1048.503,A 0.000,B 0.000,C 90.000,E1 306.537} C_DIS
LIN {X -0.222,Y -628.396,Z 1048.492,A 0.000,B 0.000,C 90.000,E1 304.532} C_DIS
LIN {X -0.042,Y -628.763,Z 1048.485,A 0.000,B 0.000,C 90.000,E1 303.245} C_DIS
LIN {X 0.155,Y -629.266,Z 1048.478,A 0.000,B 0.000,C 90.000,E1 301.957} C_DIS
LIN {X -0.143,Y -630.007,Z 1048.468,A 0.000,B 0.000,C 90.000,E1 300.207} C_DIS
LIN {X -0.255,Y -630.875,Z 1048.461,A 0.000,B 0.000,C 90.000,E1 298.949} C_DIS
LIN {X -0.196,Y -631.078,Z 1048.458,A 0.000,B 0.000,C 90.000,E1 298.437} C_DIS
LIN {X 0.163,Y -631.481,Z 1048.455,A 0.000,B 0.000,C 90.000,E1 297.897} C_DIS
LIN {X 0.227,Y -631.682,Z 1048.452,A 0.000,B 0.000,C 90.000,E1 297.385} C_DIS
LIN {X 0.259,Y -631.694,Z 1048.451,A 0.000,B 0.000,C 90.000,E1 297.129} C_DIS
LIN {X 0.293,Y -631.953,Z 1048.449,A 0.000,B 0.000,C 90.000,E1 296.873} C_DIS
LIN {X -0.137,Y -632.113,Z 1048.444,A 0.000,B 0.000,C 90.000,E1 295.899} C_DIS
LIN {X -0.104,Y -632.289,Z 1048.443,A 0.000,B 0.000,C 90.000,E1 295.643} C_DIS
LIN {X -0.306,Y -632.045,Z 1048.440,A 0.000,B 0.000,C 90.000,E1 295.155} C_DIS
LIN {X -0.238,Y -631.954,Z 1048.437,A 0.000,B 0.000,C 90.000,E1 294.643} C_DIS
LIN {X -0.205,Y -632.050,Z 1048.435,A 0.000,B 0.000,C 90.000,E1 294.387} C_DIS
LIN {X 0.242,Y -631.514,Z 1048.430,A 0.000,B 0.000,C 90.000,E1 293.334} C_DIS
LIN {X 0.080,Y -630.955,Z 1048.426,A 0.000,B 0.000,C 90.000,E1 292.589} C_DIS
LIN {X -0.068,Y -629.674,Z 1048.420,A 0.000,B 0.000,C 90.000,E1 291.589} C_DIS
LIN {X -0.052,Y -629.218,Z 1048.419,A 0.000,B 0.000,C 90.000,E1 291.334} C_DIS
LIN {X 0.333,Y -627.718,Z 1048.416,A 0.000,B 0.000,C 90.000,E1 290.791} C_DIS
LIN {X 0.119,Y -626.568,Z 1048.414,A 0.000,B 0.000,C 90.000,E1 290.556} C_DIS
LIN {X 0.121,Y -624.258,Z 1048.412,A 0.000,B 0.000,C 90.000,E1 290.174} C_DIS
LIN {X -0.100,Y -622.304,Z 1048.411,A 0.000,B 0.000,C 90.000,E1 289.939} C_DIS
LIN {X -0.115,Y -620.004,Z 1048.409,A 0.000,B 0.000,C 90.000,E1 289.685} C_DIS
LIN {X -0.331,Y -618.701,Z 1048.409,A 0.000,B 0.000,C 90.000,E1 289.577} C_DIS
LIN {X -0.143,Y -613.481,Z 1048.407,A 0.000,B 0.000,C 90.000,E1 289.214} C_DIS
LIN {X -0.282,Y -610.355,Z 1048.406,A 0.000,B 0.000,C 90.000,E1 289.033} C_DIS
LIN {X 0.031,Y -608.104,Z 1048.405,A 0.000,B 0.000,C 90.000,E1 288.906} C_DIS
LIN {X 0.085,Y -602.274,Z 1048.403,A 0.000,B 0.000,C 90.000,E1 288.598} C_DIS
LIN {X -0.116,Y -593.387,Z 1048.401,A 0.000,B 0.000,C 90.000,E1 288.236} C_DIS
LIN {X -0.174,Y -589.289,Z 1048.401,A 0.000,B 0.000,C 90.000,E1 288.109} C_DIS
LIN {X 0.003,Y -581.934,Z 1048.399,A 0.000,B 0.000,C 90.000,E1 287.873} C_DIS
LIN {X 0.103,Y -573.393,Z 1048.398,A 0.000,B 0.000,C 90.000,E1 287.638} C_DIS
LIN {X 0.196,Y -562.672,Z 1048.396,A 0.000,B 0.000,C 90.000,E1 287.330} C_DIS
LIN {X -0.246,Y -558.914,Z 1048.396,A 0.000,B 0.000,C 90.000,E1 287.275} C_DIS
LIN {X 0.161,Y -552.828,Z 1048.395,A 0.000,B 0.000,C 90.000,E1 287.040} C_DIS
LIN {X -0.092,Y -550.174,Z 1048.394,A 0.000,B 0.000,C 90.000,E1 286.913} C_DIS
LIN {X 0.084,Y -549.393,Z 1048.393,A 0.000,B 0.000,C 90.000,E1 286.804} C_DIS
LIN {X 0.073,Y -547.753,Z 1048.391,A 0.000,B 0.000,C 90.000,E1 286.441} C_DIS
LIN {X 0.221,Y -547.025,Z 1048.389,A 0.000,B 0.000,C 90.000,E1 285.898} C_DIS
LIN {X -0.122,Y -546.536,Z 1048.385,A 0.000,B 0.000,C 90.000,E1 285.371} C_DIS
LIN {X 0.180,Y -545.920,Z 1048.376,A 0.000,B 0.000,C 90.000,E1 283.647} C_DIS
LIN {X 0.101,Y -545.734,Z 1048.373,A 0.000,B 0.000,C 90.000,E1 283.175} C_DIS
LIN {X 0.060,Y -545.750,Z 1048.373,A 0.000,B 0.000,C 90.000,E1 283.175} C_DIS
LIN {X -0.165,Y -546.222,Z 1048.373,A 0.000,B 0.000,C 90.000,E1 283.119} C_DIS
LIN {X -0.072,Y -547.007,Z 1048.371,A 0.000,B 0.000,C 90.000,E1 282.827} C_DIS
LIN {X 0.025,Y -546.678,Z 1048.370,A 0.000,B 0.000,C 90.000,E1 282.535} C_DIS
LIN {X -0.037,Y -545.367,Z 1048.367,A 0.000,B 0.000,C 90.000,E1 282.119} C_DIS
LIN {X 0.149,Y -544.263,Z 1048.359,A 0.000,B 0.000,C 90.000,E1 280.546} C_DIS
LIN {X 0.043,Y -543.068,Z 1048.349,A 0.000,B 0.000,C 90.000,E1 278.859} C_DIS
LIN {X -0.175,Y -542.100,Z 1048.341,A 0.000,B 0.000,C 90.000,E1 277.466} C_DIS
LIN {X 0.058,Y -541.089,Z 1048.332,A 0.000,B 0.000,C 90.000,E1 275.739} C_DIS
LIN {X 0.216,Y -540.211,Z 1048.324,A 0.000,B 0.000,C 90.000,E1 274.302} C_DIS
LIN {X -0.154,Y -539.086,Z 1048.313,A 0.000,B 0.000,C 90.000,E1 272.350} C_DIS
LIN {X -0.052,Y -538.111,Z 1048.303,A 0.000,B 0.000,C 90.000,E1 270.630} C_DIS
LIN {X 0.016,Y -537.018,Z 1048.294,A 0.000,B 0.000,C 90.000,E1 268.912} C_DIS
LIN {X 0.066,Y -536.051,Z 1048.286,A 0.000,B 0.000,C 90.000,E1 267.478} C_DIS
LIN {X 0.094,Y -535.088,Z 1048.278,A 0.000,B 0.000,C 90.000,E1 266.045} C_DIS
LIN {X 0.157,Y -533.638,Z 1048.267,A 0.000,B 0.000,C 90.000,E1 264.033} C_DIS
LIN {X 0.213,Y -532.949,Z 1048.262,A 0.000,B 0.000,C 90.000,E1 263.166} C_DIS
LIN {X -0.223,Y -531.791,Z 1048.256,A 0.000,B 0.000,C 90.000,E1 262.064} C_DIS
LIN {X -0.155,Y -529.894,Z 1048.246,A 0.000,B 0.000,C 90.000,E1 260.330} C_DIS
LIN {X 0.015,Y -528.388,Z 1048.238,A 0.000,B 0.000,C 90.000,E1 258.870} C_DIS
LIN {X 0.159,Y -526.812,Z 1048.230,A 0.000,B 0.000,C 90.000,E1 257.409} C_DIS
LIN {X 0.051,Y -524.336,Z 1048.217,A 0.000,B 0.000,C 90.000,E1 255.102} C_DIS
LIN {X -0.133,Y -522.493,Z 1048.208,A 0.000,B 0.000,C 90.000,E1 253.378} C_DIS
LIN {X 0.136,Y -520.937,Z 1048.200,A 0.000,B 0.000,C 90.000,E1 251.891} C_DIS
LIN {X 0.204,Y -519.214,Z 1048.191,A 0.000,B 0.000,C 90.000,E1 250.423} C_DIS
LIN {X -0.142,Y -516.697,Z 1048.180,A 0.000,B 0.000,C 90.000,E1 248.411} C_DIS
LIN {X -0.217,Y -515.649,Z 1048.175,A 0.000,B 0.000,C 90.000,E1 247.539} C_DIS
LIN {X 0.071,Y -513.134,Z 1048.165,A 0.000,B 0.000,C 90.000,E1 245.741} C_DIS
LIN {X -0.071,Y -510.859,Z 1048.157,A 0.000,B 0.000,C 90.000,E1 244.280} C_DIS
LIN {X -0.023,Y -508.454,Z 1048.149,A 0.000,B 0.000,C 90.000,E1 242.794} C_DIS
LIN {X -0.017,Y -505.894,Z 1048.141,A 0.000,B 0.000,C 90.000,E1 241.307} C_DIS
LIN {X 0.182,Y -503.208,Z 1048.132,A 0.000,B 0.000,C 90.000,E1 239.793} C_DIS
LIN {X 0.189,Y -499.881,Z 1048.122,A 0.000,B 0.000,C 90.000,E1 237.995} C_DIS
LIN {X -0.183,Y -497.627,Z 1048.116,A 0.000,B 0.000,C 90.000,E1 236.834} C_DIS
LIN {X 0.100,Y -495.230,Z 1048.109,A 0.000,B 0.000,C 90.000,E1 235.595} C_DIS
LIN {X -0.062,Y -492.739,Z 1048.102,A 0.000,B 0.000,C 90.000,E1 234.402} C_DIS
LIN {X 0.110,Y -488.566,Z 1048.092,A 0.000,B 0.000,C 90.000,E1 232.557} C_DIS
LIN {X 0.094,Y -484.270,Z 1048.082,A 0.000,B 0.000,C 90.000,E1 230.723} C_DIS
LIN {X 0.289,Y -480.160,Z 1048.072,A 0.000,B 0.000,C 90.000,E1 228.852} C_DIS
LIN {X 0.234,Y -476.979,Z 1048.063,A 0.000,B 0.000,C 90.000,E1 227.310} C_DIS
LIN {X 0.068,Y -471.874,Z 1048.049,A 0.000,B 0.000,C 90.000,E1 224.838} C_DIS
LIN {X -0.082,Y -468.063,Z 1048.039,A 0.000,B 0.000,C 90.000,E1 222.975} C_DIS
LIN {X 0.044,Y -464.229,Z 1048.028,A 0.000,B 0.000,C 90.000,E1 221.067} C_DIS
LIN {X 0.038,Y -460.926,Z 1048.019,A 0.000,B 0.000,C 90.000,E1 219.483} C_DIS
LIN {X 0.036,Y -457.488,Z 1048.011,A 0.000,B 0.000,C 90.000,E1 217.890} C_DIS
LIN {X -0.028,Y -454.173,Z 1048.002,A 0.000,B 0.000,C 90.000,E1 216.297} C_DIS
LIN {X 0.026,Y -450.188,Z 1047.991,A 0.000,B 0.000,C 90.000,E1 214.358} C_DIS
LIN {X -0.010,Y -446.213,Z 1047.980,A 0.000,B 0.000,C 90.000,E1 212.418} C_DIS
LIN {X -0.068,Y -442.610,Z 1047.971,A 0.000,B 0.000,C 90.000,E1 210.797} C_DIS
LIN {X -0.041,Y -438.960,Z 1047.962,A 0.000,B 0.000,C 90.000,E1 209.155} C_DIS
LIN {X -0.109,Y -436.065,Z 1047.955,A 0.000,B 0.000,C 90.000,E1 207.847} C_DIS
LIN {X -0.025,Y -432.567,Z 1047.945,A 0.000,B 0.000,C 90.000,E1 206.181} C_DIS
LIN {X 0.125,Y -425.707,Z 1047.927,A 0.000,B 0.000,C 90.000,E1 202.823} C_DIS
LIN {X -0.046,Y -420.410,Z 1047.910,A 0.000,B 0.000,C 90.000,E1 199.812} C_DIS
LIN {X 0.036,Y -417.439,Z 1047.899,A 0.000,B 0.000,C 90.000,E1 197.764} C_DIS
LIN {X -0.100,Y -415.706,Z 1047.889,A 0.000,B 0.000,C 90.000,E1 196.079} C_DIS
LIN {X 0.010,Y -414.702,Z 1047.880,A 0.000,B 0.000,C 90.000,E1 194.356} C_DIS
LIN {X 0.187,Y -414.808,Z 1047.876,A 0.000,B 0.000,C 90.000,E1 193.647} C_DIS
LIN {X -0.135,Y -415.283,Z 1047.872,A 0.000,B 0.000,C 90.000,E1 193.008} C_DIS
LIN {X 0.047,Y -416.282,Z 1047.868,A 0.000,B 0.000,C 90.000,E1 192.299} C_DIS
LIN {X 0.096,Y -417.093,Z 1047.866,A 0.000,B 0.000,C 90.000,E1 191.951} C_DIS
LIN {X -0.191,Y -418.638,Z 1047.864,A 0.000,B 0.000,C 90.000,E1 191.478} C_DIS
LIN {X -0.061,Y -420.666,Z 1047.861,A 0.000,B 0.000,C 90.000,E1 190.950} C_DIS
LIN {X -0.202,Y -424.949,Z 1047.856,A 0.000,B 0.000,C 90.000,E1 190.141} C_DIS
LIN {X 0.062,Y -430.086,Z 1047.852,A 0.000,B 0.000,C 90.000,E1 189.265} C_DIS
LIN {X -0.089,Y -443.520,Z 1047.841,A 0.000,B 0.000,C 90.000,E1 187.296} C_DIS
LIN {X -0.003,Y -451.637,Z 1047.834,A 0.000,B 0.000,C 90.000,E1 186.144} C_DIS
LIN {X -0.173,Y -459.559,Z 1047.828,A 0.000,B 0.000,C 90.000,E1 185.049} C_DIS
LIN {X -0.215,Y -464.012,Z 1047.824,A 0.000,B 0.000,C 90.000,E1 184.416} C_DIS
LIN {X -0.111,Y -469.353,Z 1047.820,A 0.000,B 0.000,C 90.000,E1 183.612} C_DIS
LIN {X -0.148,Y -475.447,Z 1047.815,A 0.000,B 0.000,C 90.000,E1 182.694} C_DIS
LIN {X -0.219,Y -481.383,Z 1047.810,A 0.000,B 0.000,C 90.000,E1 181.776} C_DIS
LIN {X -0.023,Y -487.984,Z 1047.804,A 0.000,B 0.000,C 90.000,E1 180.688} C_DIS
LIN {X 0.202,Y -494.516,Z 1047.798,A 0.000,B 0.000,C 90.000,E1 179.599} C_DIS
LIN {X -0.219,Y -499.982,Z 1047.793,A 0.000,B 0.000,C 90.000,E1 178.740} C_DIS
LIN {X -0.179,Y -506.996,Z 1047.786,A 0.000,B 0.000,C 90.000,E1 177.535} C_DIS
LIN {X 0.183,Y -514.532,Z 1047.779,A 0.000,B 0.000,C 90.000,E1 176.159} C_DIS
LIN {X -0.094,Y -522.900,Z 1047.771,A 0.000,B 0.000,C 90.000,E1 174.723} C_DIS
LIN {X -0.172,Y -531.045,Z 1047.763,A 0.000,B 0.000,C 90.000,E1 173.280} C_DIS
LIN {X -0.100,Y -538.926,Z 1047.755,A 0.000,B 0.000,C 90.000,E1 171.837} C_DIS
LIN {X -0.075,Y -545.909,Z 1047.748,A 0.000,B 0.000,C 90.000,E1 170.557} C_DIS
LIN {X -0.193,Y -553.547,Z 1047.740,A 0.000,B 0.000,C 90.000,E1 169.162} C_DIS
LIN {X -0.073,Y -558.748,Z 1047.734,A 0.000,B 0.000,C 90.000,E1 168.173} C_DIS
LIN {X 0.005,Y -566.684,Z 1047.726,A 0.000,B 0.000,C 90.000,E1 166.645} C_DIS
LIN {X -0.026,Y -570.798,Z 1047.721,A 0.000,B 0.000,C 90.000,E1 165.825} C_DIS
LIN {X 0.220,Y -576.722,Z 1047.714,A 0.000,B 0.000,C 90.000,E1 164.574} C_DIS
LIN {X 0.189,Y -581.233,Z 1047.709,A 0.000,B 0.000,C 90.000,E1 163.630} C_DIS
LIN {X 0.217,Y -586.641,Z 1047.703,A 0.000,B 0.000,C 90.000,E1 162.417} C_DIS
LIN {X -0.024,Y -590.049,Z 1047.698,A 0.000,B 0.000,C 90.000,E1 161.638} C_DIS
LIN {X 0.203,Y -594.293,Z 1047.692,A 0.000,B 0.000,C 90.000,E1 160.550} C_DIS
LIN {X -0.075,Y -598.343,Z 1047.686,A 0.000,B 0.000,C 90.000,E1 159.518} C_DIS
LIN {X -0.004,Y -601.264,Z 1047.682,A 0.000,B 0.000,C 90.000,E1 158.720} C_DIS
LIN {X -0.040,Y -605.732,Z 1047.675,A 0.000,B 0.000,C 90.000,E1 157.411} C_DIS
LIN {X 0.052,Y -609.009,Z 1047.669,A 0.000,B 0.000,C 90.000,E1 156.357} C_DIS
LIN {X 0.146,Y -612.889,Z 1047.661,A 0.000,B 0.000,C 90.000,E1 155.049} C_DIS
LIN {X 0.053,Y -615.060,Z 1047.657,A 0.000,B 0.000,C 90.000,E1 154.280} C_DIS
LIN {X -0.031,Y -617.822,Z 1047.651,A 0.000,B 0.000,C 90.000,E1 153.256} C_DIS
LIN {X -0.082,Y -620.470,Z 1047.646,A 0.000,B 0.000,C 90.000,E1 152.231} C_DIS
LIN {X 0.196,Y -623.052,Z 1047.640,A 0.000,B 0.000,C 90.000,E1 151.179} C_DIS
LIN {X -0.015,Y -626.829,Z 1047.631,A 0.000,B 0.000,C 90.000,E1 149.665} C_DIS
LIN {X 0.169,Y -630.326,Z 1047.623,A 0.000,B 0.000,C 90.000,E1 148.122} C_DIS
LIN {X 0.037,Y -632.661,Z 1047.617,A 0.000,B 0.000,C 90.000,E1 147.120} C_DIS
LIN {X -0.233,Y -635.468,Z 1047.610,A 0.000,B 0.000,C 90.000,E1 145.881} C_DIS
LIN {X -0.073,Y -638.792,Z 1047.602,A 0.000,B 0.000,C 90.000,E1 144.356} C_DIS
LIN {X 0.010,Y -642.129,Z 1047.594,A 0.000,B 0.000,C 90.000,E1 142.844} C_DIS
LIN {X 0.077,Y -646.038,Z 1047.584,A 0.000,B 0.000,C 90.000,E1 141.090} C_DIS
LIN {X 0.285,Y -648.794,Z 1047.577,A 0.000,B 0.000,C 90.000,E1 139.828} C_DIS
LIN {X -0.009,Y -652.079,Z 1047.569,A 0.000,B 0.000,C 90.000,E1 138.366} C_DIS
LIN {X 0.164,Y -656.615,Z 1047.558,A 0.000,B 0.000,C 90.000,E1 136.377} C_DIS
LIN {X -0.028,Y -660.887,Z 1047.548,A 0.000,B 0.000,C 90.000,E1 134.676} C_DIS
LIN {X -0.120,Y -664.930,Z 1047.540,A 0.000,B 0.000,C 90.000,E1 133.218} C_DIS
LIN {X -0.107,Y -668.895,Z 1047.532,A 0.000,B 0.000,C 90.000,E1 131.757} C_DIS
LIN {X -0.016,Y -672.900,Z 1047.524,A 0.000,B 0.000,C 90.000,E1 130.297} C_DIS
LIN {X 0.234,Y -676.844,Z 1047.516,A 0.000,B 0.000,C 90.000,E1 128.830} C_DIS
LIN {X 0.007,Y -680.005,Z 1047.509,A 0.000,B 0.000,C 90.000,E1 127.649} C_DIS
LIN {X -0.202,Y -682.416,Z 1047.504,A 0.000,B 0.000,C 90.000,E1 126.710} C_DIS
LIN {X -0.009,Y -686.700,Z 1047.495,A 0.000,B 0.000,C 90.000,E1 125.025} C_DIS
LIN {X 0.260,Y -690.283,Z 1047.487,A 0.000,B 0.000,C 90.000,E1 123.579} C_DIS
LIN {X -0.229,Y -692.587,Z 1047.481,A 0.000,B 0.000,C 90.000,E1 122.673} C_DIS
LIN {X 0.126,Y -695.370,Z 1047.475,A 0.000,B 0.000,C 90.000,E1 121.465} C_DIS
LIN {X -0.079,Y -697.408,Z 1047.470,A 0.000,B 0.000,C 90.000,E1 120.541} C_DIS
LIN {X 0.438,Y -698.697,Z 1047.466,A 0.000,B 0.000,C 90.000,E1 119.795} C_DIS
LIN {X 0.272,Y -700.124,Z 1047.461,A 0.000,B 0.000,C 90.000,E1 118.871} C_DIS
LIN {X -0.212,Y -701.191,Z 1047.455,A 0.000,B 0.000,C 90.000,E1 117.975} C_DIS
LIN {X -0.114,Y -702.781,Z 1047.448,A 0.000,B 0.000,C 90.000,E1 116.565} C_DIS
LIN {X 0.384,Y -703.668,Z 1047.442,A 0.000,B 0.000,C 90.000,E1 115.591} C_DIS
LIN {X -0.058,Y -704.276,Z 1047.437,A 0.000,B 0.000,C 90.000,E1 114.695} C_DIS
LIN {X 0.217,Y -704.086,Z 1047.435,A 0.000,B 0.000,C 90.000,E1 114.207} C_DIS
LIN {X -0.142,Y -703.845,Z 1047.433,A 0.000,B 0.000,C 90.000,E1 114.003} C_DIS
LIN {X 0.135,Y -702.709,Z 1047.431,A 0.000,B 0.000,C 90.000,E1 113.515} C_DIS
LIN {X 0.135,Y -701.751,Z 1047.429,A 0.000,B 0.000,C 90.000,E1 113.281} C_DIS
LIN {X 0.034,Y -698.778,Z 1047.427,A 0.000,B 0.000,C 90.000,E1 112.823} C_DIS
LIN {X -0.106,Y -697.789,Z 1047.426,A 0.000,B 0.000,C 90.000,E1 112.717} C_DIS
LIN {X 0.026,Y -696.305,Z 1047.426,A 0.000,B 0.000,C 90.000,E1 112.589} C_DIS
LIN {X 0.259,Y -690.596,Z 1047.424,A 0.000,B 0.000,C 90.000,E1 112.280} C_DIS
LIN {X 0.204,Y -688.963,Z 1047.423,A 0.000,B 0.000,C 90.000,E1 112.206} C_DIS
LIN {X -0.084,Y -687.031,Z 1047.423,A 0.000,B 0.000,C 90.000,E1 112.153} C_DIS
LIN {X -0.113,Y -684.474,Z 1047.423,A 0.000,B 0.000,C 90.000,E1 112.078} C_DIS
LIN {X -0.157,Y -676.112,Z 1047.422,A 0.000,B 0.000,C 90.000,E1 111.972} C_DIS
LIN {X -0.200,Y -610.396,Z 1047.422,A 0.000,B 0.000,C 90.000,E1 111.972} C_DIS
LIN {X 0.208,Y -604.259,Z 1047.421,A 0.000,B 0.000,C 90.000,E1 111.716} C_DIS
LIN {X 0.018,Y -597.848,Z 1047.419,A 0.000,B 0.000,C 90.000,E1 111.408} C_DIS
LIN {X -0.070,Y -592.322,Z 1047.417,A 0.000,B 0.000,C 90.000,E1 111.046} C_DIS
LIN {X -0.084,Y -575.781,Z 1047.409,A 0.000,B 0.000,C 90.000,E1 109.704} C_DIS
LIN {X -0.243,Y -569.741,Z 1047.407,A 0.000,B 0.000,C 90.000,E1 109.268} C_DIS
LIN {X 0.170,Y -561.248,Z 1047.404,A 0.000,B 0.000,C 90.000,E1 108.725} C_DIS
LIN {X 0.209,Y -554.655,Z 1047.402,A 0.000,B 0.000,C 90.000,E1 108.362} C_DIS
LIN {X -0.024,Y -549.572,Z 1047.400,A 0.000,B 0.000,C 90.000,E1 108.055} C_DIS
LIN {X 0.251,Y -547.857,Z 1047.399,A 0.000,B 0.000,C 90.000,E1 107.819} C_DIS
LIN {X 0.209,Y -547.830,Z 1047.399,A 0.000,B 0.000,C 90.000,E1 107.819} C_DIS
LIN {X 0.168,Y -547.378,Z 1047.397,A 0.000,B 0.000,C 90.000,E1 107.511} C_DIS
LIN {X -0.075,Y -547.800,Z 1047.392,A 0.000,B 0.000,C 90.000,E1 106.551} C_DIS
LIN {X 0.258,Y -548.826,Z 1047.383,A 0.000,B 0.000,C 90.000,E1 104.828} C_DIS
LIN {X -0.155,Y -550.817,Z 1047.367,A 0.000,B 0.000,C 90.000,E1 102.063} C_DIS
LIN {X -0.052,Y -553.887,Z 1047.350,A 0.000,B 0.000,C 90.000,E1 98.973} C_DIS
LIN {X 0.100,Y -556.097,Z 1047.339,A 0.000,B 0.000,C 90.000,E1 97.004} C_DIS
LIN {X -0.210,Y -557.081,Z 1047.334,A 0.000,B 0.000,C 90.000,E1 96.201} C_DIS
LIN {X 0.178,Y -558.179,Z 1047.328,A 0.000,B 0.000,C 90.000,E1 95.049} C_DIS
LIN {X 0.021,Y -559.098,Z 1047.322,A 0.000,B 0.000,C 90.000,E1 93.955} C_DIS
LIN {X -0.079,Y -559.925,Z 1047.314,A 0.000,B 0.000,C 90.000,E1 92.579} C_DIS
LIN {X -0.256,Y -560.445,Z 1047.308,A 0.000,B 0.000,C 90.000,E1 91.489} C_DIS
LIN {X -0.248,Y -561.056,Z 1047.299,A 0.000,B 0.000,C 90.000,E1 89.828} C_DIS
LIN {X 0.235,Y -561.466,Z 1047.291,A 0.000,B 0.000,C 90.000,E1 88.396} C_DIS
LIN {X -0.260,Y -562.028,Z 1047.282,A 0.000,B 0.000,C 90.000,E1 86.788} C_DIS
LIN {X 0.252,Y -562.545,Z 1047.274,A 0.000,B 0.000,C 90.000,E1 85.355} C_DIS
LIN {X 0.244,Y -562.925,Z 1047.267,A 0.000,B 0.000,C 90.000,E1 83.976} C_DIS
LIN {X -0.256,Y -563.266,Z 1047.259,A 0.000,B 0.000,C 90.000,E1 82.648} C_DIS
LIN {X -0.272,Y -563.928,Z 1047.247,A 0.000,B 0.000,C 90.000,E1 80.443} C_DIS
LIN {X -0.002,Y -564.964,Z 1047.233,A 0.000,B 0.000,C 90.000,E1 77.937} C_DIS
LIN {X 0.029,Y -565.823,Z 1047.224,A 0.000,B 0.000,C 90.000,E1 76.284} C_DIS
LIN {X 0.252,Y -567.059,Z 1047.213,A 0.000,B 0.000,C 90.000,E1 74.338} C_DIS
LIN {X 0.309,Y -568.139,Z 1047.206,A 0.000,B 0.000,C 90.000,E1 72.960} C_DIS
LIN {X -0.194,Y -569.703,Z 1047.195,A 0.000,B 0.000,C 90.000,E1 71.094} C_DIS
LIN {X 0.087,Y -570.838,Z 1047.187,A 0.000,B 0.000,C 90.000,E1 69.699} C_DIS
LIN {X 0.026,Y -572.240,Z 1047.177,A 0.000,B 0.000,C 90.000,E1 67.794} C_DIS
LIN {X -0.315,Y -573.486,Z 1047.166,A 0.000,B 0.000,C 90.000,E1 65.921} C_DIS
LIN {X -0.074,Y -574.257,Z 1047.159,A 0.000,B 0.000,C 90.000,E1 64.537} C_DIS
LIN {X 0.272,Y -575.112,Z 1047.150,A 0.000,B 0.000,C 90.000,E1 62.871} C_DIS
LIN {X 0.124,Y -575.844,Z 1047.140,A 0.000,B 0.000,C 90.000,E1 61.257} C_DIS
LIN {X -0.236,Y -576.615,Z 1047.131,A 0.000,B 0.000,C 90.000,E1 59.665} C_DIS
LIN {X 0.227,Y -577.089,Z 1047.125,A 0.000,B 0.000,C 90.000,E1 58.535} C_DIS
LIN {X 0.040,Y -577.573,Z 1047.118,A 0.000,B 0.000,C 90.000,E1 57.199} C_DIS
LIN {X -0.314,Y -577.929,Z 1047.110,A 0.000,B 0.000,C 90.000,E1 55.881} C_DIS
LIN {X 0.148,Y -578.239,Z 1047.103,A 0.000,B 0.000,C 90.000,E1 54.482} C_DIS
LIN {X -0.015,Y -578.370,Z 1047.097,A 0.000,B 0.000,C 90.000,E1 53.417} C_DIS
LIN {X -0.180,Y -578.318,Z 1047.091,A 0.000,B 0.000,C 90.000,E1 52.351} C_DIS
LIN {X 0.006,Y -578.083,Z 1047.085,A 0.000,B 0.000,C 90.000,E1 51.251} C_DIS
LIN {X -0.099,Y -577.543,Z 1047.077,A 0.000,B 0.000,C 90.000,E1 49.908} C_DIS
LIN {X 0.163,Y -576.834,Z 1047.070,A 0.000,B 0.000,C 90.000,E1 48.528} C_DIS
LIN {X -0.115,Y -576.125,Z 1047.064,A 0.000,B 0.000,C 90.000,E1 47.472} C_DIS
LIN {X -0.020,Y -575.297,Z 1047.058,A 0.000,B 0.000,C 90.000,E1 46.377} C_DIS
LIN {X 0.058,Y -574.096,Z 1047.052,A 0.000,B 0.000,C 90.000,E1 45.283} C_DIS
LIN {X -0.003,Y -573.026,Z 1047.047,A 0.000,B 0.000,C 90.000,E1 44.474} C_DIS
LIN {X 0.042,Y -571.383,Z 1047.041,A 0.000,B 0.000,C 90.000,E1 43.380} C_DIS
LIN {X 0.067,Y -569.475,Z 1047.035,A 0.000,B 0.000,C 90.000,E1 42.285} C_DIS
LIN {X -0.004,Y -567.886,Z 1047.030,A 0.000,B 0.000,C 90.000,E1 41.472} C_DIS
LIN {X -0.032,Y -565.501,Z 1047.024,A 0.000,B 0.000,C 90.000,E1 40.378} C_DIS
LIN {X 0.071,Y -561.820,Z 1047.017,A 0.000,B 0.000,C 90.000,E1 38.991} C_DIS
LIN {X -0.070,Y -559.160,Z 1047.012,A 0.000,B 0.000,C 90.000,E1 38.177} C_DIS
LIN {X -0.243,Y -556.308,Z 1047.007,A 0.000,B 0.000,C 90.000,E1 37.363} C_DIS
LIN {X -0.081,Y -554.205,Z 1047.004,A 0.000,B 0.000,C 90.000,E1 36.790} C_DIS
LIN {X 0.064,Y -551.913,Z 1047.001,A 0.000,B 0.000,C 90.000,E1 36.217} C_DIS
LIN {X -0.019,Y -546.981,Z 1046.995,A 0.000,B 0.000,C 90.000,E1 35.105} C_DIS
LIN {X -0.070,Y -543.582,Z 1046.991,A 0.000,B 0.000,C 90.000,E1 34.405} C_DIS
LIN {X -0.133,Y -538.388,Z 1046.986,A 0.000,B 0.000,C 90.000,E1 33.420} C_DIS
LIN {X 0.039,Y -535.299,Z 1046.982,A 0.000,B 0.000,C 90.000,E1 32.832} C_DIS
LIN {X 0.155,Y -528.515,Z 1046.976,A 0.000,B 0.000,C 90.000,E1 31.671} C_DIS
LIN {X 0.056,Y -521.988,Z 1046.970,A 0.000,B 0.000,C 90.000,E1 30.669} C_DIS
LIN {X -0.046,Y -516.910,Z 1046.966,A 0.000,B 0.000,C 90.000,E1 29.951} C_DIS
LIN {X 0.234,Y -512.516,Z 1046.963,A 0.000,B 0.000,C 90.000,E1 29.333} C_DIS
LIN {X 0.123,Y -504.125,Z 1046.957,A 0.000,B 0.000,C 90.000,E1 28.309} C_DIS
LIN {X -0.043,Y -497.462,Z 1046.953,A 0.000,B 0.000,C 90.000,E1 27.590} C_DIS
LIN {X 0.111,Y -490.796,Z 1046.949,A 0.000,B 0.000,C 90.000,E1 26.873} C_DIS
LIN {X -0.051,Y -483.819,Z 1046.945,A 0.000,B 0.000,C 90.000,E1 26.181} C_DIS
LIN {X 0.131,Y -472.547,Z 1046.939,A 0.000,B 0.000,C 90.000,E1 25.079} C_DIS
LIN {X -0.264,Y -462.374,Z 1046.934,A 0.000,B 0.000,C 90.000,E1 24.207} C_DIS
LIN {X 0.066,Y -451.619,Z 1046.929,A 0.000,B 0.000,C 90.000,E1 23.259} C_DIS
LIN {X 0.016,Y -427.934,Z 1046.918,A 0.000,B 0.000,C 90.000,E1 21.153} C_DIS
LIN {X -0.144,Y -417.911,Z 1046.912,A 0.000,B 0.000,C 90.000,E1 20.174} C_DIS
LIN {X -0.149,Y -406.825,Z 1046.905,A 0.000,B 0.000,C 90.000,E1 18.960} C_DIS
LIN {X -0.100,Y -399.114,Z 1046.900,A 0.000,B 0.000,C 90.000,E1 18.000} C_DIS
LIN {X 0.141,Y -396.019,Z 1046.897,A 0.000,B 0.000,C 90.000,E1 17.511} C_DIS
LIN {X 0.060,Y -395.018,Z 1046.896,A 0.000,B 0.000,C 90.000,E1 17.347} C_DIS
LIN {X 0.012,Y -393.023,Z 1046.894,A 0.000,B 0.000,C 90.000,E1 16.913} C_DIS
LIN {X -0.063,Y -391.737,Z 1046.891,A 0.000,B 0.000,C 90.000,E1 16.386} C_DIS
LIN {X 0.033,Y -391.443,Z 1046.887,A 0.000,B 0.000,C 90.000,E1 15.662} C_DIS
LIN {X 0.200,Y -391.756,Z 1046.884,A 0.000,B 0.000,C 90.000,E1 15.064} C_DIS
LIN {X -0.036,Y -398.687,Z 1046.854,A 0.000,B 0.000,C 90.000,E1 9.792} C_DIS
LIN {X 0.210,Y -405.919,Z 1046.833,A 0.000,B 0.000,C 90.000,E1 5.910} C_DIS
LIN {X 0.136,Y -409.687,Z 1046.823,A 0.000,B 0.000,C 90.000,E1 4.188} C_DIS
LIN {X 0.131,Y -411.732,Z 1046.819,A 0.000,B 0.000,C 90.000,E1 3.326} C_DIS
LIN {X 0.035,Y -414.098,Z 1046.815,A 0.000,B 0.000,C 90.000,E1 2.751} C_DIS
LIN {X 0.035,Y -415.023,Z 1046.814,A 0.000,B 0.000,C 90.000,E1 2.579} C_DIS
LIN {X -0.119,Y -417.435,Z 1046.812,A 0.000,B 0.000,C 90.000,E1 2.236} C_DIS
LIN {X -0.057,Y -420.668,Z 1046.811,A 0.000,B 0.000,C 90.000,E1 1.892} C_DIS
LIN {X -0.102,Y -422.008,Z 1046.810,A 0.000,B 0.000,C 90.000,E1 1.776} C_DIS
LIN {X 0.075,Y -434.162,Z 1046.806,A 0.000,B 0.000,C 90.000,E1 0.974} C_DIS
LIN {X 0.171,Y -453.039,Z 1046.799,A 0.000,B 0.000,C 90.000,E1 359.771} C_DIS
LIN {X 0.134,Y -472.894,Z 1046.792,A 0.000,B 0.000,C 90.000,E1 358.568} C_DIS
LIN {X -0.081,Y -487.473,Z 1046.787,A 0.000,B 0.000,C 90.000,E1 357.707} C_DIS
LIN {X 0.132,Y -497.140,Z 1046.784,A 0.000,B 0.000,C 90.000,E1 357.078} C_DIS
LIN {X 0.096,Y -504.973,Z 1046.781,A 0.000,B 0.000,C 90.000,E1 356.560} C_DIS
LIN {X -0.193,Y -511.153,Z 1046.779,A 0.000,B 0.000,C 90.000,E1 356.159} C_DIS
LIN {X -0.104,Y -517.342,Z 1046.776,A 0.000,B 0.000,C 90.000,E1 355.698} C_DIS
LIN {X -0.162,Y -524.586,Z 1046.773,A 0.000,B 0.000,C 90.000,E1 355.122} C_DIS
LIN {X -0.019,Y -531.661,Z 1046.769,A 0.000,B 0.000,C 90.000,E1 354.489} C_DIS
LIN {X -0.156,Y -538.387,Z 1046.766,A 0.000,B 0.000,C 90.000,E1 353.856} C_DIS
LIN {X -0.080,Y -544.841,Z 1046.762,A 0.000,B 0.000,C 90.000,E1 353.166} C_DIS
LIN {X -0.099,Y -550.714,Z 1046.758,A 0.000,B 0.000,C 90.000,E1 352.470} C_DIS
LIN {X 0.097,Y -555.045,Z 1046.755,A 0.000,B 0.000,C 90.000,E1 351.894} C_DIS
LIN {X 0.151,Y -559.801,Z 1046.751,A 0.000,B 0.000,C 90.000,E1 351.197} C_DIS
LIN {X 0.203,Y -564.124,Z 1046.747,A 0.000,B 0.000,C 90.000,E1 350.500} C_DIS
LIN {X 0.292,Y -568.081,Z 1046.744,A 0.000,B 0.000,C 90.000,E1 349.803} C_DIS
LIN {X 0.046,Y -573.141,Z 1046.738,A 0.000,B 0.000,C 90.000,E1 348.870} C_DIS
LIN {X 0.091,Y -577.096,Z 1046.734,A 0.000,B 0.000,C 90.000,E1 348.049} C_DIS
LIN {X -0.061,Y -581.295,Z 1046.728,A 0.000,B 0.000,C 90.000,E1 347.117} C_DIS
LIN {X -0.134,Y -585.844,Z 1046.722,A 0.000,B 0.000,C 90.000,E1 346.047} C_DIS
LIN {X -0.190,Y -592.108,Z 1046.714,A 0.000,B 0.000,C 90.000,E1 344.448} C_DIS
LIN {X -0.106,Y -596.127,Z 1046.708,A 0.000,B 0.000,C 90.000,E1 343.378} C_DIS
LIN {X -0.251,Y -598.992,Z 1046.703,A 0.000,B 0.000,C 90.000,E1 342.598} C_DIS
LIN {X -0.179,Y -603.410,Z 1046.696,A 0.000,B 0.000,C 90.000,E1 341.275} C_DIS
LIN {X -0.056,Y -605.862,Z 1046.692,A 0.000,B 0.000,C 90.000,E1 340.477} C_DIS
LIN {X -0.176,Y -608.941,Z 1046.686,A 0.000,B 0.000,C 90.000,E1 339.444} C_DIS
LIN {X -0.262,Y -611.721,Z 1046.680,A 0.000,B 0.000,C 90.000,E1 338.411} C_DIS
LIN {X -0.123,Y -614.999,Z 1046.673,A 0.000,B 0.000,C 90.000,E1 337.102} C_DIS
LIN {X 0.075,Y -617.937,Z 1046.666,A 0.000,B 0.000,C 90.000,E1 335.793} C_DIS
LIN {X -0.247,Y -620.457,Z 1046.658,A 0.000,B 0.000,C 90.000,E1 334.537} C_DIS
LIN {X -0.263,Y -622.181,Z 1046.653,A 0.000,B 0.000,C 90.000,E1 333.512} C_DIS
LIN {X -0.255,Y -623.802,Z 1046.647,A 0.000,B 0.000,C 90.000,E1 332.487} C_DIS
LIN {X 0.058,Y -624.943,Z 1046.643,A 0.000,B 0.000,C 90.000,E1 331.691} C_DIS
LIN {X 0.106,Y -626.514,Z 1046.636,A 0.000,B 0.000,C 90.000,E1 330.411} C_DIS
LIN {X 0.251,Y -627.763,Z 1046.629,A 0.000,B 0.000,C 90.000,E1 329.125} C_DIS
LIN {X 0.099,Y -628.838,Z 1046.622,A 0.000,B 0.000,C 90.000,E1 327.867} C_DIS
LIN {X 0.115,Y -629.531,Z 1046.613,A 0.000,B 0.000,C 90.000,E1 326.342} C_DIS
LIN {X -0.046,Y -629.730,Z 1046.607,A 0.000,B 0.000,C 90.000,E1 325.341} C_DIS
LIN {X -0.015,Y -629.789,Z 1046.600,A 0.000,B 0.000,C 90.000,E1 324.069} C_DIS
LIN {X 0.035,Y -629.718,Z 1046.595,A 0.000,B 0.000,C 90.000,E1 323.050} C_DIS
LIN {X -0.376,Y -629.760,Z 1046.582,A 0.000,B 0.000,C 90.000,E1 320.803} C_DIS
LIN {X -0.228,Y -629.909,Z 1046.572,A 0.000,B 0.000,C 90.000,E1 319.013} C_DIS
LIN {X -0.034,Y -629.892,Z 1046.558,A 0.000,B 0.000,C 90.000,E1 316.458} C_DIS
LIN {X -0.055,Y -629.943,Z 1046.552,A 0.000,B 0.000,C 90.000,E1 315.445} C_DIS
LIN {X -0.312,Y -630.025,Z 1046.544,A 0.000,B 0.000,C 90.000,E1 313.947} C_DIS
LIN {X -0.213,Y -630.108,Z 1046.534,A 0.000,B 0.000,C 90.000,E1 312.162} C_DIS
LIN {X 0.130,Y -630.007,Z 1046.527,A 0.000,B 0.000,C 90.000,E1 310.862} C_DIS
LIN {X -0.422,Y -629.984,Z 1046.520,A 0.000,B 0.000,C 90.000,E1 309.644} C_DIS
LIN {X 0.029,Y -629.868,Z 1046.514,A 0.000,B 0.000,C 90.000,E1 308.588} C_DIS
LIN {X 0.275,Y -629.824,Z 1046.505,A 0.000,B 0.000,C 90.000,E1 306.790} C_DIS
LIN {X 0.112,Y -629.727,Z 1046.502,A 0.000,B 0.000,C 90.000,E1 306.297} C_DIS
LIN {X -0.049,Y -629.786,Z 1046.499,A 0.000,B 0.000,C 90.000,E1 305.804} C_DIS
LIN {X 0.193,Y -630.331,Z 1046.485,A 0.000,B 0.000,C 90.000,E1 303.245} C_DIS
LIN {X -0.118,Y -630.869,Z 1046.478,A 0.000,B 0.000,C 90.000,E1 302.005} C_DIS
LIN {X 0.156,Y -631.695,Z 1046.468,A 0.000,B 0.000,C 90.000,E1 300.207} C_DIS
LIN {X 0.107,Y -632.718,Z 1046.459,A 0.000,B 0.000,C 90.000,E1 298.693} C_DIS
LIN {X 0.142,Y -632.815,Z 1046.458,A 0.000,B 0.000,C 90.000,E1 298.437} C_DIS
LIN {X 0.180,Y -633.103,Z 1046.457,A 0.000,B 0.000,C 90.000,E1 298.180} C_DIS
LIN {X 0.104,Y -633.804,Z 1046.450,A 0.000,B 0.000,C 90.000,E1 296.924} C_DIS
LIN {X -0.099,Y -633.940,Z 1046.447,A 0.000,B 0.000,C 90.000,E1 296.437} C_DIS
LIN {X -0.056,Y -634.161,Z 1046.445,A 0.000,B 0.000,C 90.000,E1 296.181} C_DIS
LIN {X 0.029,Y -634.226,Z 1046.443,A 0.000,B 0.000,C 90.000,E1 295.668} C_DIS
LIN {X 0.115,Y -634.120,Z 1046.440,A 0.000,B 0.000,C 90.000,E1 295.155} C_DIS
LIN {X 0.156,Y -634.229,Z 1046.438,A 0.000,B 0.000,C 90.000,E1 294.899} C_DIS
LIN {X 0.057,Y -633.962,Z 1046.433,A 0.000,B 0.000,C 90.000,E1 293.898} C_DIS
LIN {X -0.044,Y -633.449,Z 1046.427,A 0.000,B 0.000,C 90.000,E1 292.898} C_DIS
LIN {X -0.187,Y -632.820,Z 1046.423,A 0.000,B 0.000,C 90.000,E1 292.153} C_DIS
LIN {X -0.338,Y -631.910,Z 1046.419,A 0.000,B 0.000,C 90.000,E1 291.408} C_DIS
LIN {X 0.275,Y -631.278,Z 1046.417,A 0.000,B 0.000,C 90.000,E1 291.099} C_DIS
LIN {X 0.088,Y -629.573,Z 1046.415,A 0.000,B 0.000,C 90.000,E1 290.610} C_DIS
LIN {X -0.110,Y -626.729,Z 1046.412,A 0.000,B 0.000,C 90.000,E1 290.120} C_DIS
LIN {X -0.109,Y -625.841,Z 1046.411,A 0.000,B 0.000,C 90.000,E1 289.993} C_DIS
LIN {X -0.221,Y -620.781,Z 1046.408,A 0.000,B 0.000,C 90.000,E1 289.504} C_DIS
LIN {X -0.383,Y -619.038,Z 1046.408,A 0.000,B 0.000,C 90.000,E1 289.396} C_DIS
LIN {X 0.155,Y -612.925,Z 1046.406,A 0.000,B 0.000,C 90.000,E1 288.960} C_DIS
LIN {X -0.308,Y -610.815,Z 1046.405,A 0.000,B 0.000,C 90.000,E1 288.906} C_DIS
LIN {X -0.122,Y -606.867,Z 1046.404,A 0.000,B 0.000,C 90.000,E1 288.725} C_DIS
LIN {X 0.205,Y -603.988,Z 1046.403,A 0.000,B 0.000,C 90.000,E1 288.544} C_DIS
LIN {X -0.107,Y -602.063,Z 1046.403,A 0.000,B 0.000,C 90.000,E1 288.489} C_DIS
LIN {X -0.308,Y -598.200,Z 1046.402,A 0.000,B 0.000,C 90.000,E1 288.362} C_DIS
LIN {X -0.309,Y -593.940,Z 1046.401,A 0.000,B 0.000,C 90.000,E1 288.181} C_DIS
LIN {X -0.177,Y -584.468,Z 1046.399,A 0.000,B 0.000,C 90.000,E1 287.873} C_DIS
LIN {X -0.155,Y -573.966,Z 1046.398,A 0.000,B 0.000,C 90.000,E1 287.583} C_DIS
LIN {X -0.128,Y -565.458,Z 1046.396,A 0.000,B 0.000,C 90.000,E1 287.330} C_DIS
LIN {X -0.159,Y -555.394,Z 1046.394,A 0.000,B 0.000,C 90.000,E1 286.968} C_DIS
LIN {X 0.044,Y -550.623,Z 1046.393,A 0.000,B 0.000,C 90.000,E1 286.677} C_DIS
LIN {X -0.012,Y -550.571,Z 1046.393,A 0.000,B 0.000,C 90.000,E1 286.677} C_DIS
LIN {X 0.007,Y -548.911,Z 1046.391,A 0.000,B 0.000,C 90.000,E1 286.386} C_DIS
LIN {X -0.128,Y -548.354,Z 1046.390,A 0.000,B 0.000,C 90.000,E1 286.260} C_DIS
LIN {X 0.099,Y -547.142,Z 1046.385,A 0.000,B 0.000,C 90.000,E1 285.300} C_DIS
LIN {X 0.019,Y -546.286,Z 1046.375,A 0.000,B 0.000,C 90.000,E1 283.411} C_DIS
LIN {X -0.023,Y -546.298,Z 1046.375,A 0.000,B 0.000,C 90.000,E1 283.411} C_DIS
LIN {X 0.213,Y -547.490,Z 1046.373,A 0.000,B 0.000,C 90.000,E1 283.175} C_DIS
LIN {X -0.069,Y -548.114,Z 1046.373,A 0.000,B 0.000,C 90.000,E1 283.063} C_DIS
LIN {X 0.033,Y -548.755,Z 1046.371,A 0.000,B 0.000,C 90.000,E1 282.771} C_DIS
LIN {X 0.136,Y -548.383,Z 1046.370,A 0.000,B 0.000,C 90.000,E1 282.479} C_DIS
LIN {X -0.020,Y -547.757,Z 1046.369,A 0.000,B 0.000,C 90.000,E1 282.355} C_DIS
LIN {X -0.293,Y -546.918,Z 1046.368,A 0.000,B 0.000,C 90.000,E1 282.243} C_DIS
LIN {X 0.110,Y -545.818,Z 1046.366,A 0.000,B 0.000,C 90.000,E1 281.951} C_DIS
LIN {X 0.094,Y -545.006,Z 1046.361,A 0.000,B 0.000,C 90.000,E1 280.894} C_DIS
LIN {X 0.170,Y -543.200,Z 1046.348,A 0.000,B 0.000,C 90.000,E1 278.624} C_DIS
LIN {X 0.031,Y -541.707,Z 1046.335,A 0.000,B 0.000,C 90.000,E1 276.372} C_DIS
LIN {X 0.199,Y -540.837,Z 1046.328,A 0.000,B 0.000,C 90.000,E1 274.935} C_DIS
LIN {X -0.169,Y -539.812,Z 1046.318,A 0.000,B 0.000,C 90.000,E1 273.269} C_DIS
LIN {X -0.061,Y -539.004,Z 1046.310,A 0.000,B 0.000,C 90.000,E1 271.835} C_DIS
LIN {X 0.013,Y -538.373,Z 1046.304,A 0.000,B 0.000,C 90.000,E1 270.688} C_DIS
LIN {X 0.087,Y -537.260,Z 1046.294,A 0.000,B 0.000,C 90.000,E1 268.969} C_DIS
LIN {X 0.141,Y -536.305,Z 1046.286,A 0.000,B 0.000,C 90.000,E1 267.535} C_DIS
LIN {X 0.175,Y -535.313,Z 1046.278,A 0.000,B 0.000,C 90.000,E1 266.102} C_DIS
LIN {X 0.246,Y -533.861,Z 1046.267,A 0.000,B 0.000,C 90.000,E1 264.090} C_DIS
LIN {X -0.184,Y -532.912,Z 1046.261,A 0.000,B 0.000,C 90.000,E1 262.989} C_DIS
